LIN {X 0,Y 136.603,Z 356.091,A -85,B 0,C 180,E1 -24831.12,E2 -24831.12} C_VEL
LIN {X 0,Y 137.128,Z 356.027,A -85,B 0,C 180,E1 -24839.999,E2 -24839.999} C_VEL
LIN {X 0,Y 136.602,Z 356.09,A -85,B 0,C 180,E1 -24848.878,E2 -24848.878} C_VEL
LIN {X 0,Y 136.486,Z 356.105,A -85,B 0,C 180,E1 -24851.958,E2 -24851.958} C_VEL
LIN {X 0,Y 136.245,Z 356.134,A -85,B 0,C 180,E1 -24858.028,E2 -24858.028} C_VEL
LIN {X 0,Y 136.192,Z 356.144,A -85,B 0,C 180,E1 -24861.749,E2 -24861.749} C_VEL
LIN {X 0,Y 136.144,Z 356.148,A -85,B 0,C 180,E1 -24868.655,E2 -24868.655} C_VEL
LIN {X 0,Y 136.524,Z 356.287,A -85,B 0,C 180,E1 -24874.892,E2 -24874.892} C_VEL
LIN {X 0,Y 137.979,Z 362.492,A -85,B 0,C 180,E1 -24881.464,E2 -24881.464} C_VEL
LIN {X 0,Y 139.435,Z 367.911,A -85,B 0,C 180,E1 -24886.957,E2 -24886.957} C_VEL
LIN {X 0,Y 139.496,Z 370.039,A -85,B 0,C 180,E1 -24889.087,E2 -24889.087} C_VEL
LIN {X 0,Y 138.032,Z 374.626,A -85,B 0,C 180,E1 -24893.623,E2 -24893.623} C_VEL
LIN {X 0,Y 137.72,Z 379.074,A -85,B 0,C 180,E1 -24894.305,E2 -24894.305} C_VEL
LIN {X 0,Y 137.356,Z 394.701,A -85,B 0,C 180,E1 -24896.634,E2 -24896.634} C_VEL
LIN {X 0,Y 137.591,Z 410.054,A -85,B 0,C 180,E1 -24899.558,E2 -24899.558} C_VEL
LIN {X 0,Y 138.336,Z 425.298,A -85,B 0,C 180,E1 -24903.159,E2 -24903.159} C_VEL
LIN {X 0,Y 139.367,Z 438.842,A -85,B 0,C 180,E1 -24906.998,E2 -24906.998} C_VEL
LIN {X 0,Y 140.321,Z 447.525,A -85,B 0,C 180,E1 -24909.862,E2 -24909.862} C_VEL
LIN {X 0,Y 139.234,Z 457.776,A -85,B 0,C 180,E1 -24914.111,E2 -24914.111} C_VEL
LIN {X 0,Y 138.787,Z 467.552,A -85,B 0,C 180,E1 -24919.056,E2 -24919.056} C_VEL
LIN {X 0,Y 139.313,Z 475.809,A -85,B 0,C 180,E1 -24924.212,E2 -24924.212} C_VEL
LIN {X 0,Y 140.282,Z 481.655,A -85,B 0,C 180,E1 -24928.711,E2 -24928.711} C_VEL
LIN {X 0,Y 140.568,Z 483.669,A -85,B 0,C 180,E1 -24930.647,E2 -24930.647} C_VEL
LIN {X 0,Y 139.909,Z 485.281,A -85,B 0,C 180,E1 -24932.882,E2 -24932.882} C_VEL
LIN {X 0,Y 137.869,Z 488.121,A -85,B 0,C 180,E1 -24938.799,E2 -24938.799} C_VEL
LIN {X 0,Y 137.224,Z 489.871,A -85,B 0,C 180,E1 -24944.84,E2 -24944.84} C_VEL
LIN {X 0,Y 138.316,Z 490.738,A -85,B 0,C 180,E1 -24950.838,E2 -24950.838} C_VEL
LIN {X 0,Y 141.251,Z 490.873,A -85,B 0,C 180,E1 -24956.605,E2 -24956.605} C_VEL
LIN {X 0,Y 148.821,Z 489.76,A -85,B 0,C 180,E1 -24964.523,E2 -24964.523} C_VEL
LIN {X 0,Y 159.675,Z 487.114,A -85,B 0,C 180,E1 -24971.319,E2 -24971.319} C_VEL
LIN {X 0,Y 168.489,Z 484.531,A -85,B 0,C 180,E1 -24975.165,E2 -24975.165} C_VEL
LIN {X 0,Y 181.11,Z 480.199,A -85,B 0,C 180,E1 -24979.582,E2 -24979.582} C_VEL
LIN {X 0,Y 181.549,Z 479.751,A -85,B 0,C 180,E1 -24980.201,E2 -24980.201} C_VEL
LIN {X 0,Y 174.225,Z 479.446,A -85,B 0,C 180,E1 -24982.766,E2 -24982.766} C_VEL
LIN {X 0,Y 162.472,Z 477.5,A -85,B 0,C 180,E1 -24987.929,E2 -24987.929} C_VEL
LIN {X 0,Y 154.17,Z 474.585,A -85,B 0,C 180,E1 -24992.88,E2 -24992.88} C_VEL
LIN {X 0,Y 147.888,Z 470.965,A -85,B 0,C 180,E1 -24997.702,E2 -24997.702} C_VEL
LIN {X 0,Y 145.198,Z 469.279,A -85,B 0,C 180,E1 -24999.639,E2 -24999.639} C_VEL
LIN {X 0,Y 139.454,Z 466.109,A -85,B 0,C 180,E1 -25002.635,E2 -25002.635} C_VEL
LIN {X 0,Y 134.168,Z 462.429,A -85,B 0,C 180,E1 -25005.808,E2 -25005.808} C_VEL
LIN {X 0,Y 132.282,Z 459.913,A -85,B 0,C 180,E1 -25007.973,E2 -25007.973} C_VEL
LIN {X 0,Y 129.903,Z 451.969,A -85,B 0,C 180,E1 -25014.568,E2 -25014.568} C_VEL
LIN {X 0,Y 129.082,Z 443.16,A -85,B 0,C 180,E1 -25020.781,E2 -25020.781} C_VEL
LIN {X 0,Y 129.146,Z 432.525,A -85,B 0,C 180,E1 -25027.034,E2 -25027.034} C_VEL
LIN {X 0,Y 130.087,Z 423.208,A -85,B 0,C 180,E1 -25031.69,E2 -25031.69} C_VEL
LIN {X 0,Y 131.579,Z 412.383,A -85,B 0,C 180,E1 -25036.286,E2 -25036.286} C_VEL
LIN {X 0,Y 133.527,Z 399.543,A -85,B 0,C 180,E1 -25040.811,E2 -25040.811} C_VEL
LIN {X 0,Y 135.909,Z 385.871,A -85,B 0,C 180,E1 -25044.78,E2 -25044.78} C_VEL
LIN {X 0,Y 135.967,Z 384.573,A -85,B 0,C 180,E1 -25045.112,E2 -25045.112} C_VEL
LIN {X 0,Y 132.484,Z 371.01,A -85,B 0,C 180,E1 -25048.519,E2 -25048.519} C_VEL
LIN {X 0,Y 129.268,Z 357.522,A -85,B 0,C 180,E1 -25051.607,E2 -25051.607} C_VEL
LIN {X 0,Y 129.144,Z 357.047,A -85,B 0,C 180,E1 -25052.223,E2 -25052.223} C_VEL
LIN {X 0,Y 128.941,Z 357.043,A -85,B 0,C 180,E1 -25056.84,E2 -25056.84} C_VEL
LIN {X 0,Y 128.951,Z 357.047,A -85,B 0,C 180,E1 -25060.847,E2 -25060.847} C_VEL
LIN {X 0,Y 128.931,Z 357.043,A -85,B 0,C 180,E1 -25065.125,E2 -25065.125} C_VEL
LIN {X 0,Y 128.965,Z 357.045,A -85,B 0,C 180,E1 -25069.725,E2 -25069.725} C_VEL
LIN {X 0,Y 128.998,Z 357.038,A -85,B 0,C 180,E1 -25074.809,E2 -25074.809} C_VEL
LIN {X 0,Y 129.022,Z 357.034,A -85,B 0,C 180,E1 -25080.64,E2 -25080.64} C_VEL
LIN {X 0,Y 129.032,Z 357.035,A -85,B 0,C 180,E1 -25084.165,E2 -25084.165} C_VEL
LIN {X 0,Y 129.112,Z 357.027,A -85,B 0,C 180,E1 -25087.726,E2 -25087.726} C_VEL
LIN {X 0,Y 129.164,Z 357.014,A -85,B 0,C 180,E1 -25090.943,E2 -25090.943} C_VEL
LIN {X 0,Y 129.423,Z 356.985,A -85,B 0,C 180,E1 -25097.813,E2 -25097.813} C_VEL
LIN {X 0,Y 129.536,Z 356.971,A -85,B 0,C 180,E1 -25100.63,E2 -25100.63} C_VEL
LIN {X 0,Y 130.094,Z 356.903,A -85,B 0,C 180,E1 -25109.997,E2 -25109.997} C_VEL
LIN {X 0,Y 129.534,Z 356.974,A -85,B 0,C 180,E1 -25119.365,E2 -25119.365} C_VEL
LIN {X 0,Y 129.397,Z 356.99,A -85,B 0,C 180,E1 -25122.545,E2 -25122.545} C_VEL
LIN {X 0,Y 129.165,Z 357.021,A -85,B 0,C 180,E1 -25129.051,E2 -25129.051} C_VEL
LIN {X 0,Y 129.109,Z 357.023,A -85,B 0,C 180,E1 -25132.395,E2 -25132.395} C_VEL
LIN {X 0,Y 129.031,Z 357.036,A -85,B 0,C 180,E1 -25135.829,E2 -25135.829} C_VEL
LIN {X 0,Y 129.016,Z 357.038,A -85,B 0,C 180,E1 -25139.355,E2 -25139.355} C_VEL
LIN {X 0,Y 128.98,Z 357.043,A -85,B 0,C 180,E1 -25145.18,E2 -25145.18} C_VEL
LIN {X 0,Y 128.932,Z 357.043,A -85,B 0,C 180,E1 -25150.848,E2 -25150.848} C_VEL
LIN {X 0,Y 128.918,Z 357.052,A -85,B 0,C 180,E1 -25155.124,E2 -25155.124} C_VEL
LIN {X 0,Y 128.939,Z 357.043,A -85,B 0,C 180,E1 -25159.732,E2 -25159.732} C_VEL
LIN {X 0,Y 128.979,Z 357.044,A -85,B 0,C 180,E1 -25164.814,E2 -25164.814} C_VEL
LIN {X 0,Y 129.046,Z 357.034,A -85,B 0,C 180,E1 -25170.649,E2 -25170.649} C_VEL
LIN {X 0,Y 129.103,Z 357.025,A -85,B 0,C 180,E1 -25177.725,E2 -25177.725} C_VEL
LIN {X 0,Y 129.158,Z 357.022,A -85,B 0,C 180,E1 -25180.944,E2 -25180.944} C_VEL
LIN {X 0,Y 129.413,Z 356.988,A -85,B 0,C 180,E1 -25187.813,E2 -25187.813} C_VEL
LIN {X 0,Y 129.525,Z 356.975,A -85,B 0,C 180,E1 -25190.631,E2 -25190.631} C_VEL
LIN {X 0,Y 130.084,Z 356.905,A -85,B 0,C 180,E1 -25199.999,E2 -25199.999} C_VEL
LIN {X 0,Y 129.524,Z 356.971,A -85,B 0,C 180,E1 -25209.368,E2 -25209.368} C_VEL
LIN {X 0,Y 129.388,Z 356.992,A -85,B 0,C 180,E1 -25212.548,E2 -25212.548} C_VEL
LIN {X 0,Y 129.153,Z 357.014,A -85,B 0,C 180,E1 -25219.055,E2 -25219.055} C_VEL
LIN {X 0,Y 129.102,Z 357.029,A -85,B 0,C 180,E1 -25222.399,E2 -25222.399} C_VEL
LIN {X 0,Y 129.097,Z 357.026,A -85,B 0,C 180,E1 -25229.427,E2 -25229.427} C_VEL
LIN {X 0,Y 129.494,Z 357.096,A -85,B 0,C 180,E1 -25235.283,E2 -25235.283} C_VEL
LIN {X 0,Y 130.801,Z 362.398,A -85,B 0,C 180,E1 -25241.221,E2 -25241.221} C_VEL
LIN {X 0,Y 132.11,Z 367.066,A -85,B 0,C 180,E1 -25246.25,E2 -25246.25} C_VEL
LIN {X 0,Y 132.475,Z 368.687,A -85,B 0,C 180,E1 -25247.963,E2 -25247.963} C_VEL
LIN {X 0,Y 131.943,Z 370.854,A -85,B 0,C 180,E1 -25250.273,E2 -25250.273} C_VEL
LIN {X 0,Y 131.065,Z 373.682,A -85,B 0,C 180,E1 -25253.166,E2 -25253.166} C_VEL
LIN {X 0,Y 130.265,Z 391.666,A -85,B 0,C 180,E1 -25255.965,E2 -25255.965} C_VEL
LIN {X 0,Y 130.43,Z 406.961,A -85,B 0,C 180,E1 -25258.967,E2 -25258.967} C_VEL
LIN {X 0,Y 131.047,Z 421.405,A -85,B 0,C 180,E1 -25262.451,E2 -25262.451} C_VEL
LIN {X 0,Y 132.042,Z 435.246,A -85,B 0,C 180,E1 -25266.476,E2 -25266.476} C_VEL
LIN {X 0,Y 133.341,Z 446.662,A -85,B 0,C 180,E1 -25270.369,E2 -25270.369} C_VEL
LIN {X 0,Y 132.394,Z 456.294,A -85,B 0,C 180,E1 -25274.611,E2 -25274.611} C_VEL
LIN {X 0,Y 132.062,Z 465.103,A -85,B 0,C 180,E1 -25279.268,E2 -25279.268} C_VEL
LIN {X 0,Y 132.653,Z 473.561,A -85,B 0,C 180,E1 -25284.683,E2 -25284.683} C_VEL
LIN {X 0,Y 133.563,Z 478.708,A -85,B 0,C 180,E1 -25288.73,E2 -25288.73} C_VEL
LIN {X 0,Y 133.876,Z 480.168,A -85,B 0,C 180,E1 -25290.003,E2 -25290.003} C_VEL
LIN {X 0,Y 133.296,Z 482.552,A -85,B 0,C 180,E1 -25293.025,E2 -25293.025} C_VEL
LIN {X 0,Y 131.23,Z 485.546,A -85,B 0,C 180,E1 -25299.248,E2 -25299.248} C_VEL
LIN {X 0,Y 130.635,Z 487.479,A -85,B 0,C 180,E1 -25305.607,E2 -25305.607} C_VEL
LIN {X 0,Y 131.911,Z 488.565,A -85,B 0,C 180,E1 -25311.9,E2 -25311.9} C_VEL
LIN {X 0,Y 135.079,Z 488.926,A -85,B 0,C 180,E1 -25317.924,E2 -25317.924} C_VEL
LIN {X 0,Y 140.013,Z 488.576,A -85,B 0,C 180,E1 -25323.517,E2 -25323.517} C_VEL
LIN {X 0,Y 146.563,Z 487.63,A -85,B 0,C 180,E1 -25328.566,E2 -25328.566} C_VEL
LIN {X 0,Y 158.864,Z 484.979,A -85,B 0,C 180,E1 -25335.061,E2 -25335.061} C_VEL
LIN {X 0,Y 171.356,Z 481.571,A -85,B 0,C 180,E1 -25339.656,E2 -25339.656} C_VEL
LIN {X 0,Y 170.756,Z 481.068,A -85,B 0,C 180,E1 -25340.61,E2 -25340.61} C_VEL
LIN {X 0,Y 159.635,Z 479.231,A -85,B 0,C 180,E1 -25345.088,E2 -25345.088} C_VEL
LIN {X 0,Y 151.563,Z 476.711,A -85,B 0,C 180,E1 -25349.332,E2 -25349.332} C_VEL
LIN {X 0,Y 142.923,Z 472.226,A -85,B 0,C 180,E1 -25355.294,E2 -25355.294} C_VEL
LIN {X 0,Y 136.232,Z 466.215,A -85,B 0,C 180,E1 -25361.97,E2 -25361.97} C_VEL
LIN {X 0,Y 132.282,Z 459.913,A -85,B 0,C 180,E1 -25367.973,E2 -25367.973} C_VEL
LIN {X 0,Y 130.663,Z 457.299,A -85,B 0,C 180,E1 -25370.158,E2 -25370.158} C_VEL
LIN {X 0,Y 126.723,Z 452.536,A -85,B 0,C 180,E1 -25373.598,E2 -25373.598} C_VEL
LIN {X 0,Y 123.152,Z 447.252,A -85,B 0,C 180,E1 -25377.117,E2 -25377.117} C_VEL
LIN {X 0,Y 122.177,Z 443.872,A -85,B 0,C 180,E1 -25379.36,E2 -25379.36} C_VEL
LIN {X 0,Y 121.971,Z 433.547,A -85,B 0,C 180,E1 -25385.788,E2 -25385.788} C_VEL
LIN {X 0,Y 122.985,Z 423.193,A -85,B 0,C 180,E1 -25391.256,E2 -25391.256} C_VEL
LIN {X 0,Y 124.542,Z 411.592,A -85,B 0,C 180,E1 -25396.39,E2 -25396.39} C_VEL
LIN {X 0,Y 126.539,Z 398.546,A -85,B 0,C 180,E1 -25401.163,E2 -25401.163} C_VEL
LIN {X 0,Y 128.82,Z 385.674,A -85,B 0,C 180,E1 -25405.013,E2 -25405.013} C_VEL
LIN {X 0,Y 125.748,Z 373.225,A -85,B 0,C 180,E1 -25408.323,E2 -25408.323} C_VEL
LIN {X 0,Y 122.197,Z 358.436,A -85,B 0,C 180,E1 -25411.898,E2 -25411.898} C_VEL
LIN {X 0,Y 122.095,Z 357.915,A -85,B 0,C 180,E1 -25412.658,E2 -25412.658} C_VEL
LIN {X 0,Y 121.87,Z 357.928,A -85,B 0,C 180,E1 -25419.373,E2 -25419.373} C_VEL
LIN {X 0,Y 121.855,Z 357.928,A -85,B 0,C 180,E1 -25423.798,E2 -25423.798} C_VEL
LIN {X 0,Y 121.892,Z 357.927,A -85,B 0,C 180,E1 -25428.553,E2 -25428.553} C_VEL
LIN {X 0,Y 121.951,Z 357.915,A -85,B 0,C 180,E1 -25434.806,E2 -25434.806} C_VEL
LIN {X 0,Y 121.935,Z 357.92,A -85,B 0,C 180,E1 -25439.835,E2 -25439.835} C_VEL
LIN {X 0,Y 121.987,Z 357.916,A -85,B 0,C 180,E1 -25446.213,E2 -25446.213} C_VEL
LIN {X 0,Y 122.054,Z 357.901,A -85,B 0,C 180,E1 -25449.785,E2 -25449.785} C_VEL
LIN {X 0,Y 122.269,Z 357.878,A -85,B 0,C 180,E1 -25456.705,E2 -25456.705} C_VEL
LIN {X 0,Y 122.462,Z 357.85,A -85,B 0,C 180,E1 -25460.083,E2 -25460.083} C_VEL
LIN {X 0,Y 122.614,Z 357.832,A -85,B 0,C 180,E1 -25466.711,E2 -25466.711} C_VEL
LIN {X 0,Y 123.048,Z 357.781,A -85,B 0,C 180,E1 -25469.997,E2 -25469.997} C_VEL
LIN {X 0,Y 122.459,Z 357.849,A -85,B 0,C 180,E1 -25476.588,E2 -25476.588} C_VEL
LIN {X 0,Y 122.46,Z 357.856,A -85,B 0,C 180,E1 -25479.911,E2 -25479.911} C_VEL
LIN {X 0,Y 122.267,Z 357.877,A -85,B 0,C 180,E1 -25483.289,E2 -25483.289} C_VEL
LIN {X 0,Y 122.053,Z 357.905,A -85,B 0,C 180,E1 -25490.208,E2 -25490.208} C_VEL
LIN {X 0,Y 121.984,Z 357.909,A -85,B 0,C 180,E1 -25493.781,E2 -25493.781} C_VEL
LIN {X 0,Y 121.928,Z 357.919,A -85,B 0,C 180,E1 -25500.16,E2 -25500.16} C_VEL
LIN {X 0,Y 121.898,Z 357.925,A -85,B 0,C 180,E1 -25506.178,E2 -25506.178} C_VEL
LIN {X 0,Y 121.87,Z 357.924,A -85,B 0,C 180,E1 -25511.436,E2 -25511.436} C_VEL
LIN {X 0,Y 121.869,Z 357.924,A -85,B 0,C 180,E1 -25518.558,E2 -25518.558} C_VEL
LIN {X 0,Y 121.931,Z 357.921,A -85,B 0,C 180,E1 -25524.802,E2 -25524.802} C_VEL
LIN {X 0,Y 121.937,Z 357.918,A -85,B 0,C 180,E1 -25529.824,E2 -25529.824} C_VEL
LIN {X 0,Y 121.979,Z 357.909,A -85,B 0,C 180,E1 -25536.213,E2 -25536.213} C_VEL
LIN {X 0,Y 122.046,Z 357.906,A -85,B 0,C 180,E1 -25539.786,E2 -25539.786} C_VEL
LIN {X 0,Y 122.26,Z 357.878,A -85,B 0,C 180,E1 -25546.706,E2 -25546.706} C_VEL
LIN {X 0,Y 122.451,Z 357.857,A -85,B 0,C 180,E1 -25550.084,E2 -25550.084} C_VEL
LIN {X 0,Y 122.605,Z 357.838,A -85,B 0,C 180,E1 -25556.713,E2 -25556.713} C_VEL
LIN {X 0,Y 123.038,Z 357.782,A -85,B 0,C 180,E1 -25559.999,E2 -25559.999} C_VEL
LIN {X 0,Y 122.45,Z 357.857,A -85,B 0,C 180,E1 -25566.591,E2 -25566.591} C_VEL
LIN {X 0,Y 122.45,Z 357.851,A -85,B 0,C 180,E1 -25569.914,E2 -25569.914} C_VEL
LIN {X 0,Y 122.258,Z 357.879,A -85,B 0,C 180,E1 -25573.293,E2 -25573.293} C_VEL
LIN {X 0,Y 122.043,Z 357.903,A -85,B 0,C 180,E1 -25580.213,E2 -25580.213} C_VEL
LIN {X 0,Y 121.978,Z 357.917,A -85,B 0,C 180,E1 -25583.785,E2 -25583.785} C_VEL
LIN {X 0,Y 122.078,Z 357.903,A -85,B 0,C 180,E1 -25591.206,E2 -25591.206} C_VEL
LIN {X 0,Y 122.496,Z 357.946,A -85,B 0,C 180,E1 -25595.868,E2 -25595.868} C_VEL
LIN {X 0,Y 124.059,Z 363.872,A -85,B 0,C 180,E1 -25602.828,E2 -25602.828} C_VEL
LIN {X 0,Y 125.274,Z 368.163,A -85,B 0,C 180,E1 -25607.689,E2 -25607.689} C_VEL
LIN {X 0,Y 124.989,Z 369.943,A -85,B 0,C 180,E1 -25609.716,E2 -25609.716} C_VEL
LIN {X 0,Y 124.089,Z 372.745,A -85,B 0,C 180,E1 -25612.704,E2 -25612.704} C_VEL
LIN {X 0,Y 123.219,Z 389.789,A -85,B 0,C 180,E1 -25615.491,E2 -25615.491} C_VEL
LIN {X 0,Y 123.305,Z 405.547,A -85,B 0,C 180,E1 -25618.753,E2 -25618.753} C_VEL
LIN {X 0,Y 123.878,Z 418.797,A -85,B 0,C 180,E1 -25622.096,E2 -25622.096} C_VEL
LIN {X 0,Y 124.848,Z 432.037,A -85,B 0,C 180,E1 -25626.073,E2 -25626.073} C_VEL
LIN {X 0,Y 126.355,Z 444.58,A -85,B 0,C 180,E1 -25630.508,E2 -25630.508} C_VEL
LIN {X 0,Y 125.677,Z 453.596,A -85,B 0,C 180,E1 -25634.599,E2 -25634.599} C_VEL
LIN {X 0,Y 125.369,Z 462.556,A -85,B 0,C 180,E1 -25639.506,E2 -25639.506} C_VEL
LIN {X 0,Y 126.046,Z 471.181,A -85,B 0,C 180,E1 -25645.205,E2 -25645.205} C_VEL
LIN {X 0,Y 127.183,Z 477.053,A -85,B 0,C 180,E1 -25650.003,E2 -25650.003} C_VEL
LIN {X 0,Y 127.128,Z 479.003,A -85,B 0,C 180,E1 -25652.137,E2 -25652.137} C_VEL
LIN {X 0,Y 125.538,Z 481.421,A -85,B 0,C 180,E1 -25656.432,E2 -25656.432} C_VEL
LIN {X 0,Y 124.145,Z 484.024,A -85,B 0,C 180,E1 -25663.091,E2 -25663.091} C_VEL
LIN {X 0,Y 125.566,Z 486.272,A -85,B 0,C 180,E1 -25673.069,E2 -25673.069} C_VEL
LIN {X 0,Y 131.414,Z 486.873,A -85,B 0,C 180,E1 -25682.333,E2 -25682.333} C_VEL
LIN {X 0,Y 141.162,Z 486.044,A -85,B 0,C 180,E1 -25690.336,E2 -25690.336} C_VEL
LIN {X 0,Y 151.835,Z 484.281,A -85,B 0,C 180,E1 -25696.029,E2 -25696.029} C_VEL
LIN {X 0,Y 160.67,Z 482.448,A -85,B 0,C 180,E1 -25699.412,E2 -25699.412} C_VEL
LIN {X 0,Y 161.702,Z 481.829,A -85,B 0,C 180,E1 -25700.417,E2 -25700.417} C_VEL
LIN {X 0,Y 149.542,Z 478.811,A -85,B 0,C 180,E1 -25705.671,E2 -25705.671} C_VEL
LIN {X 0,Y 139.9,Z 474.457,A -85,B 0,C 180,E1 -25711.495,E2 -25711.495} C_VEL
LIN {X 0,Y 132.089,Z 468.633,A -85,B 0,C 180,E1 -25718.134,E2 -25718.134} C_VEL
LIN {X 0,Y 127.318,Z 462.817,A -85,B 0,C 180,E1 -25723.979,E2 -25723.979} C_VEL
LIN {X 0,Y 124.094,Z 455.854,A -85,B 0,C 180,E1 -25730.219,E2 -25730.219} C_VEL
LIN {X 0,Y 122.424,Z 447.597,A -85,B 0,C 180,E1 -25736.71,E2 -25736.71} C_VEL
LIN {X 0,Y 122.177,Z 443.872,A -85,B 0,C 180,E1 -25739.36,E2 -25739.36} C_VEL
LIN {X 0,Y 121.347,Z 440.448,A -85,B 0,C 180,E1 -25741.551,E2 -25741.551} C_VEL
LIN {X 0,Y 118.608,Z 434.253,A -85,B 0,C 180,E1 -25744.993,E2 -25744.993} C_VEL
LIN {X 0,Y 116.159,Z 427.641,A -85,B 0,C 180,E1 -25748.439,E2 -25748.439} C_VEL
LIN {X 0,Y 115.837,Z 423.476,A -85,B 0,C 180,E1 -25750.559,E2 -25750.559} C_VEL
LIN {X 0,Y 117.373,Z 411.494,A -85,B 0,C 180,E1 -25756.155,E2 -25756.155} C_VEL
LIN {X 0,Y 119.409,Z 398.529,A -85,B 0,C 180,E1 -25761.132,E2 -25761.132} C_VEL
LIN {X 0,Y 121.588,Z 385.463,A -85,B 0,C 180,E1 -25765.233,E2 -25765.233} C_VEL
LIN {X 0,Y 117.891,Z 370.949,A -85,B 0,C 180,E1 -25769.229,E2 -25769.229} C_VEL
LIN {X 0,Y 115.161,Z 359.392,A -85,B 0,C 180,E1 -25772.124,E2 -25772.124} C_VEL
LIN {X 0,Y 115.043,Z 358.81,A -85,B 0,C 180,E1 -25772.806,E2 -25772.806} C_VEL
LIN {X 0,Y 114.795,Z 358.806,A -85,B 0,C 180,E1 -25777.752,E2 -25777.752} C_VEL
LIN {X 0,Y 114.799,Z 358.808,A -85,B 0,C 180,E1 -25782.719,E2 -25782.719} C_VEL
LIN {X 0,Y 114.811,Z 358.807,A -85,B 0,C 180,E1 -25787.67,E2 -25787.67} C_VEL
LIN {X 0,Y 114.818,Z 358.801,A -85,B 0,C 180,E1 -25792.726,E2 -25792.726} C_VEL
LIN {X 0,Y 114.869,Z 358.8,A -85,B 0,C 180,E1 -25798.934,E2 -25798.934} C_VEL
LIN {X 0,Y 114.952,Z 358.791,A -85,B 0,C 180,E1 -25806.505,E2 -25806.505} C_VEL
LIN {X 0,Y 115.023,Z 358.778,A -85,B 0,C 180,E1 -25812.208,E2 -25812.208} C_VEL
LIN {X 0,Y 115.291,Z 358.747,A -85,B 0,C 180,E1 -25817.255,E2 -25817.255} C_VEL
LIN {X 0,Y 115.398,Z 358.728,A -85,B 0,C 180,E1 -25819.469,E2 -25819.469} C_VEL
LIN {X 0,Y 115.541,Z 358.713,A -85,B 0,C 180,E1 -25826.51,E2 -25826.51} C_VEL
LIN {X 0,Y 116,Z 358.658,A -85,B 0,C 180,E1 -25829.997,E2 -25829.997} C_VEL
LIN {X 0,Y 115.401,Z 358.728,A -85,B 0,C 180,E1 -25836.993,E2 -25836.993} C_VEL
LIN {X 0,Y 115.396,Z 358.735,A -85,B 0,C 180,E1 -25840.524,E2 -25840.524} C_VEL
LIN {X 0,Y 115.151,Z 358.76,A -85,B 0,C 180,E1 -25844.127,E2 -25844.127} C_VEL
LIN {X 0,Y 114.985,Z 358.784,A -85,B 0,C 180,E1 -25851.51,E2 -25851.51} C_VEL
LIN {X 0,Y 114.868,Z 358.798,A -85,B 0,C 180,E1 -25855.355,E2 -25855.355} C_VEL
LIN {X 0,Y 114.861,Z 358.797,A -85,B 0,C 180,E1 -25861.059,E2 -25861.059} C_VEL
LIN {X 0,Y 114.787,Z 358.81,A -85,B 0,C 180,E1 -25867.749,E2 -25867.749} C_VEL
LIN {X 0,Y 114.785,Z 358.809,A -85,B 0,C 180,E1 -25872.714,E2 -25872.714} C_VEL
LIN {X 0,Y 114.792,Z 358.807,A -85,B 0,C 180,E1 -25877.664,E2 -25877.664} C_VEL
LIN {X 0,Y 114.796,Z 358.81,A -85,B 0,C 180,E1 -25882.733,E2 -25882.733} C_VEL
LIN {X 0,Y 114.864,Z 358.797,A -85,B 0,C 180,E1 -25888.93,E2 -25888.93} C_VEL
LIN {X 0,Y 114.942,Z 358.785,A -85,B 0,C 180,E1 -25896.505,E2 -25896.505} C_VEL
LIN {X 0,Y 115.015,Z 358.783,A -85,B 0,C 180,E1 -25902.209,E2 -25902.209} C_VEL
LIN {X 0,Y 115.281,Z 358.749,A -85,B 0,C 180,E1 -25907.256,E2 -25907.256} C_VEL
LIN {X 0,Y 115.387,Z 358.736,A -85,B 0,C 180,E1 -25909.471,E2 -25909.471} C_VEL
LIN {X 0,Y 115.531,Z 358.719,A -85,B 0,C 180,E1 -25916.511,E2 -25916.511} C_VEL
LIN {X 0,Y 115.99,Z 358.659,A -85,B 0,C 180,E1 -25919.999,E2 -25919.999} C_VEL
LIN {X 0,Y 115.391,Z 358.735,A -85,B 0,C 180,E1 -25926.996,E2 -25926.996} C_VEL
LIN {X 0,Y 115.387,Z 358.73,A -85,B 0,C 180,E1 -25930.528,E2 -25930.528} C_VEL
LIN {X 0,Y 115.142,Z 358.768,A -85,B 0,C 180,E1 -25934.131,E2 -25934.131} C_VEL
LIN {X 0,Y 114.975,Z 358.786,A -85,B 0,C 180,E1 -25941.515,E2 -25941.515} C_VEL
LIN {X 0,Y 114.945,Z 358.788,A -85,B 0,C 180,E1 -25949.283,E2 -25949.283} C_VEL
LIN {X 0,Y 115.542,Z 358.831,A -85,B 0,C 180,E1 -25956.644,E2 -25956.644} C_VEL
LIN {X 0,Y 117.198,Z 364.745,A -85,B 0,C 180,E1 -25963.983,E2 -25963.983} C_VEL
LIN {X 0,Y 118.061,Z 367.502,A -85,B 0,C 180,E1 -25967.275,E2 -25967.275} C_VEL
LIN {X 0,Y 117.979,Z 368.975,A -85,B 0,C 180,E1 -25969.064,E2 -25969.064} C_VEL
LIN {X 0,Y 117.129,Z 371.717,A -85,B 0,C 180,E1 -25972.185,E2 -25972.185} C_VEL
LIN {X 0,Y 116.125,Z 390.044,A -85,B 0,C 180,E1 -25975.436,E2 -25975.436} C_VEL
LIN {X 0,Y 116.21,Z 405.08,A -85,B 0,C 180,E1 -25978.793,E2 -25978.793} C_VEL
LIN {X 0,Y 116.886,Z 419.636,A -85,B 0,C 180,E1 -25982.777,E2 -25982.777} C_VEL
LIN {X 0,Y 118.001,Z 433.198,A -85,B 0,C 180,E1 -25987.227,E2 -25987.227} C_VEL
LIN {X 0,Y 119.468,Z 443.707,A -85,B 0,C 180,E1 -25991.217,E2 -25991.217} C_VEL
LIN {X 0,Y 118.867,Z 452.41,A -85,B 0,C 180,E1 -25995.45,E2 -25995.45} C_VEL
LIN {X 0,Y 118.728,Z 461.287,A -85,B 0,C 180,E1 -26000.635,E2 -26000.635} C_VEL
LIN {X 0,Y 119.631,Z 469.815,A -85,B 0,C 180,E1 -26006.635,E2 -26006.635} C_VEL
LIN {X 0,Y 120.512,Z 473.84,A -85,B 0,C 180,E1 -26010.003,E2 -26010.003} C_VEL
LIN {X 0,Y 120.619,Z 476.129,A -85,B 0,C 180,E1 -26012.488,E2 -26012.488} C_VEL
LIN {X 0,Y 119.014,Z 478.497,A -85,B 0,C 180,E1 -26016.786,E2 -26016.786} C_VEL
LIN {X 0,Y 117.643,Z 481.293,A -85,B 0,C 180,E1 -26023.828,E2 -26023.828} C_VEL
LIN {X 0,Y 118.248,Z 483.15,A -85,B 0,C 180,E1 -26030.895,E2 -26030.895} C_VEL
LIN {X 0,Y 120.971,Z 484.318,A -85,B 0,C 180,E1 -26037.699,E2 -26037.699} C_VEL
LIN {X 0,Y 128.691,Z 484.775,A -85,B 0,C 180,E1 -26046.925,E2 -26046.925} C_VEL
LIN {X 0,Y 140.063,Z 483.886,A -85,B 0,C 180,E1 -26054.63,E2 -26054.63} C_VEL
LIN {X 0,Y 150.91,Z 482.32,A -85,B 0,C 180,E1 -26059.501,E2 -26059.501} C_VEL
LIN {X 0,Y 151.707,Z 481.773,A -85,B 0,C 180,E1 -26060.553,E2 -26060.553} C_VEL
LIN {X 0,Y 143.768,Z 479.307,A -85,B 0,C 180,E1 -26064.084,E2 -26064.084} C_VEL
LIN {X 0,Y 133.714,Z 474.546,A -85,B 0,C 180,E1 -26070.046,E2 -26070.046} C_VEL
LIN {X 0,Y 125.537,Z 468.298,A -85,B 0,C 180,E1 -26076.929,E2 -26076.929} C_VEL
LIN {X 0,Y 120.534,Z 462.141,A -85,B 0,C 180,E1 -26083.051,E2 -26083.051} C_VEL
LIN {X 0,Y 116.899,Z 453.816,A -85,B 0,C 180,E1 -26090.484,E2 -26090.484} C_VEL
LIN {X 0,Y 115.298,Z 443.812,A -85,B 0,C 180,E1 -26098.254,E2 -26098.254} C_VEL
LIN {X 0,Y 114.952,Z 433.045,A -85,B 0,C 180,E1 -26105.263,E2 -26105.263} C_VEL
LIN {X 0,Y 115.837,Z 423.476,A -85,B 0,C 180,E1 -26110.559,E2 -26110.559} C_VEL
LIN {X 0,Y 115.61,Z 419.264,A -85,B 0,C 180,E1 -26112.602,E2 -26112.602} C_VEL
LIN {X 0,Y 113.739,Z 411.934,A -85,B 0,C 180,E1 -26115.794,E2 -26115.794} C_VEL
LIN {X 0,Y 112.043,Z 404.218,A -85,B 0,C 180,E1 -26118.888,E2 -26118.888} C_VEL
LIN {X 0,Y 112.118,Z 399.429,A -85,B 0,C 180,E1 -26120.694,E2 -26120.694} C_VEL
LIN {X 0,Y 114.346,Z 386.674,A -85,B 0,C 180,E1 -26124.997,E2 -26124.997} C_VEL
LIN {X 0,Y 113.506,Z 382.445,A -85,B 0,C 180,E1 -26126.29,E2 -26126.29} C_VEL
LIN {X 0,Y 109.686,Z 367.249,A -85,B 0,C 180,E1 -26130.516,E2 -26130.516} C_VEL
LIN {X 0,Y 108.121,Z 360.193,A -85,B 0,C 180,E1 -26132.427,E2 -26132.427} C_VEL
LIN {X 0,Y 107.978,Z 359.683,A -85,B 0,C 180,E1 -26133.188,E2 -26133.188} C_VEL
LIN {X 0,Y 107.693,Z 359.696,A -85,B 0,C 180,E1 -26140.739,E2 -26140.739} C_VEL
LIN {X 0,Y 107.691,Z 359.689,A -85,B 0,C 180,E1 -26145.88,E2 -26145.88} C_VEL
LIN {X 0,Y 107.715,Z 359.691,A -85,B 0,C 180,E1 -26151.534,E2 -26151.534} C_VEL
LIN {X 0,Y 107.808,Z 359.681,A -85,B 0,C 180,E1 -26158.562,E2 -26158.562} C_VEL
LIN {X 0,Y 107.917,Z 359.667,A -85,B 0,C 180,E1 -26166.996,E2 -26166.996} C_VEL
LIN {X 0,Y 108.045,Z 359.651,A -85,B 0,C 180,E1 -26174.915,E2 -26174.915} C_VEL
LIN {X 0,Y 108.311,Z 359.611,A -85,B 0,C 180,E1 -26178.772,E2 -26178.772} C_VEL
LIN {X 0,Y 108.467,Z 359.594,A -85,B 0,C 180,E1 -26186.282,E2 -26186.282} C_VEL
LIN {X 0,Y 108.951,Z 359.536,A -85,B 0,C 180,E1 -26189.997,E2 -26189.997} C_VEL
LIN {X 0,Y 108.343,Z 359.608,A -85,B 0,C 180,E1 -26197.451,E2 -26197.451} C_VEL
LIN {X 0,Y 108.205,Z 359.629,A -85,B 0,C 180,E1 -26203.022,E2 -26203.022} C_VEL
LIN {X 0,Y 107.912,Z 359.668,A -85,B 0,C 180,E1 -26209,E2 -26209} C_VEL
LIN {X 0,Y 107.857,Z 359.669,A -85,B 0,C 180,E1 -26214.18,E2 -26214.18} C_VEL
LIN {X 0,Y 107.787,Z 359.676,A -85,B 0,C 180,E1 -26222.042,E2 -26222.042} C_VEL
LIN {X 0,Y 107.694,Z 359.693,A -85,B 0,C 180,E1 -26228.452,E2 -26228.452} C_VEL
LIN {X 0,Y 107.674,Z 359.697,A -85,B 0,C 180,E1 -26235.883,E2 -26235.883} C_VEL
LIN {X 0,Y 107.693,Z 359.694,A -85,B 0,C 180,E1 -26241.541,E2 -26241.541} C_VEL
LIN {X 0,Y 107.801,Z 359.675,A -85,B 0,C 180,E1 -26248.562,E2 -26248.562} C_VEL
LIN {X 0,Y 107.906,Z 359.662,A -85,B 0,C 180,E1 -26256.996,E2 -26256.996} C_VEL
LIN {X 0,Y 108.035,Z 359.646,A -85,B 0,C 180,E1 -26264.916,E2 -26264.916} C_VEL
LIN {X 0,Y 108.301,Z 359.62,A -85,B 0,C 180,E1 -26268.773,E2 -26268.773} C_VEL
LIN {X 0,Y 108.457,Z 359.599,A -85,B 0,C 180,E1 -26276.284,E2 -26276.284} C_VEL
LIN {X 0,Y 108.941,Z 359.537,A -85,B 0,C 180,E1 -26279.999,E2 -26279.999} C_VEL
LIN {X 0,Y 108.334,Z 359.615,A -85,B 0,C 180,E1 -26287.454,E2 -26287.454} C_VEL
LIN {X 0,Y 108.197,Z 359.631,A -85,B 0,C 180,E1 -26293.025,E2 -26293.025} C_VEL
LIN {X 0,Y 107.902,Z 359.661,A -85,B 0,C 180,E1 -26299.005,E2 -26299.005} C_VEL
LIN {X 0,Y 107.856,Z 359.675,A -85,B 0,C 180,E1 -26304.191,E2 -26304.191} C_VEL
LIN {X 0,Y 108.04,Z 359.652,A -85,B 0,C 180,E1 -26312.266,E2 -26312.266} C_VEL
LIN {X 0,Y 108.641,Z 359.723,A -85,B 0,C 180,E1 -26317.626,E2 -26317.626} C_VEL
LIN {X 0,Y 110.199,Z 364.975,A -85,B 0,C 180,E1 -26324.549,E2 -26324.549} C_VEL
LIN {X 0,Y 110.947,Z 367.679,A -85,B 0,C 180,E1 -26327.989,E2 -26327.989} C_VEL
LIN {X 0,Y 110.184,Z 370.692,A -85,B 0,C 180,E1 -26331.696,E2 -26331.696} C_VEL
LIN {X 0,Y 109.166,Z 386.383,A -85,B 0,C 180,E1 -26334.595,E2 -26334.595} C_VEL
LIN {X 0,Y 109.04,Z 400.994,A -85,B 0,C 180,E1 -26337.957,E2 -26337.957} C_VEL
LIN {X 0,Y 109.663,Z 416.43,A -85,B 0,C 180,E1 -26342.317,E2 -26342.317} C_VEL
LIN {X 0,Y 110.74,Z 429.214,A -85,B 0,C 180,E1 -26346.635,E2 -26346.635} C_VEL
LIN {X 0,Y 112.507,Z 442.211,A -85,B 0,C 180,E1 -26351.804,E2 -26351.804} C_VEL
LIN {X 0,Y 112.286,Z 447.785,A -85,B 0,C 180,E1 -26354.577,E2 -26354.577} C_VEL
LIN {X 0,Y 112.057,Z 457.192,A -85,B 0,C 180,E1 -26360.072,E2 -26360.072} C_VEL
LIN {X 0,Y 112.925,Z 466.188,A -85,B 0,C 180,E1 -26366.435,E2 -26366.435} C_VEL
LIN {X 0,Y 113.816,Z 470.443,A -85,B 0,C 180,E1 -26370.003,E2 -26370.003} C_VEL
LIN {X 0,Y 114.214,Z 472.258,A -85,B 0,C 180,E1 -26371.766,E2 -26371.766} C_VEL
LIN {X 0,Y 113.862,Z 473.566,A -85,B 0,C 180,E1 -26373.542,E2 -26373.542} C_VEL
LIN {X 0,Y 111.664,Z 477.082,A -85,B 0,C 180,E1 -26380.887,E2 -26380.887} C_VEL
LIN {X 0,Y 111.998,Z 480.493,A -85,B 0,C 180,E1 -26392.121,E2 -26392.121} C_VEL
LIN {X 0,Y 117.303,Z 482.264,A -85,B 0,C 180,E1 -26402.634,E2 -26402.634} C_VEL
LIN {X 0,Y 126.895,Z 482.626,A -85,B 0,C 180,E1 -26411.656,E2 -26411.656} C_VEL
LIN {X 0,Y 139.831,Z 481.709,A -85,B 0,C 180,E1 -26418.934,E2 -26418.934} C_VEL
LIN {X 0,Y 142.798,Z 481.338,A -85,B 0,C 180,E1 -26420.223,E2 -26420.223} C_VEL
LIN {X 0,Y 131.61,Z 476.68,A -85,B 0,C 180,E1 -26425.896,E2 -26425.896} C_VEL
LIN {X 0,Y 122.164,Z 470.621,A -85,B 0,C 180,E1 -26432.599,E2 -26432.599} C_VEL
LIN {X 0,Y 115.007,Z 462.971,A -85,B 0,C 180,E1 -26440.361,E2 -26440.361} C_VEL
LIN {X 0,Y 110.637,Z 454.587,A -85,B 0,C 180,E1 -26448.087,E2 -26448.087} C_VEL
LIN {X 0,Y 108.511,Z 444.582,A -85,B 0,C 180,E1 -26456.287,E2 -26456.287} C_VEL
LIN {X 0,Y 107.908,Z 435.279,A -85,B 0,C 180,E1 -26462.801,E2 -26462.801} C_VEL
LIN {X 0,Y 108.636,Z 424.474,A -85,B 0,C 180,E1 -26469.309,E2 -26469.309} C_VEL
LIN {X 0,Y 110.033,Z 412.553,A -85,B 0,C 180,E1 -26475.289,E2 -26475.289} C_VEL
LIN {X 0,Y 112.118,Z 399.429,A -85,B 0,C 180,E1 -26480.694,E2 -26480.694} C_VEL
LIN {X 0,Y 112.201,Z 396.281,A -85,B 0,C 180,E1 -26481.835,E2 -26481.835} C_VEL
LIN {X 0,Y 111.185,Z 391.443,A -85,B 0,C 180,E1 -26483.493,E2 -26483.493} C_VEL
LIN {X 0,Y 109.323,Z 386.676,A -85,B 0,C 180,E1 -26485.052,E2 -26485.052} C_VEL
LIN {X 0,Y 106.336,Z 380.026,A -85,B 0,C 180,E1 -26487.159,E2 -26487.159} C_VEL
LIN {X 0,Y 103.819,Z 373.119,A -85,B 0,C 180,E1 -26489.233,E2 -26489.233} C_VEL
LIN {X 0,Y 101.045,Z 361.082,A -85,B 0,C 180,E1 -26492.655,E2 -26492.655} C_VEL
LIN {X 0,Y 100.905,Z 360.579,A -85,B 0,C 180,E1 -26493.295,E2 -26493.295} C_VEL
LIN {X 0,Y 100.653,Z 360.571,A -85,B 0,C 180,E1 -26499.814,E2 -26499.814} C_VEL
LIN {X 0,Y 100.661,Z 360.564,A -85,B 0,C 180,E1 -26505.714,E2 -26505.714} C_VEL
LIN {X 0,Y 100.652,Z 360.57,A -85,B 0,C 180,E1 -26511.062,E2 -26511.062} C_VEL
LIN {X 0,Y 100.704,Z 360.566,A -85,B 0,C 180,E1 -26516.876,E2 -26516.876} C_VEL
LIN {X 0,Y 100.791,Z 360.554,A -85,B 0,C 180,E1 -26525.265,E2 -26525.265} C_VEL
LIN {X 0,Y 100.824,Z 360.545,A -85,B 0,C 180,E1 -26529.599,E2 -26529.599} C_VEL
LIN {X 0,Y 101.204,Z 360.498,A -85,B 0,C 180,E1 -26537.972,E2 -26537.972} C_VEL
LIN {X 0,Y 101.284,Z 360.492,A -85,B 0,C 180,E1 -26542.019,E2 -26542.019} C_VEL
LIN {X 0,Y 101.875,Z 360.417,A -85,B 0,C 180,E1 -26549.996,E2 -26549.996} C_VEL
LIN {X 0,Y 101.282,Z 360.489,A -85,B 0,C 180,E1 -26557.974,E2 -26557.974} C_VEL
LIN {X 0,Y 101.131,Z 360.508,A -85,B 0,C 180,E1 -26563.36,E2 -26563.36} C_VEL
LIN {X 0,Y 100.821,Z 360.55,A -85,B 0,C 180,E1 -26570.394,E2 -26570.394} C_VEL
LIN {X 0,Y 100.774,Z 360.552,A -85,B 0,C 180,E1 -26574.954,E2 -26574.954} C_VEL
LIN {X 0,Y 100.694,Z 360.561,A -85,B 0,C 180,E1 -26583.115,E2 -26583.115} C_VEL
LIN {X 0,Y 100.643,Z 360.567,A -85,B 0,C 180,E1 -26589.811,E2 -26589.811} C_VEL
LIN {X 0,Y 100.645,Z 360.572,A -85,B 0,C 180,E1 -26595.708,E2 -26595.708} C_VEL
LIN {X 0,Y 100.63,Z 360.571,A -85,B 0,C 180,E1 -26601.055,E2 -26601.055} C_VEL
LIN {X 0,Y 100.693,Z 360.56,A -85,B 0,C 180,E1 -26606.875,E2 -26606.875} C_VEL
LIN {X 0,Y 100.781,Z 360.55,A -85,B 0,C 180,E1 -26615.264,E2 -26615.264} C_VEL
LIN {X 0,Y 100.814,Z 360.551,A -85,B 0,C 180,E1 -26619.599,E2 -26619.599} C_VEL
LIN {X 0,Y 101.193,Z 360.504,A -85,B 0,C 180,E1 -26627.973,E2 -26627.973} C_VEL
LIN {X 0,Y 101.273,Z 360.49,A -85,B 0,C 180,E1 -26632.021,E2 -26632.021} C_VEL
LIN {X 0,Y 101.865,Z 360.418,A -85,B 0,C 180,E1 -26639.999,E2 -26639.999} C_VEL
LIN {X 0,Y 101.273,Z 360.493,A -85,B 0,C 180,E1 -26647.977,E2 -26647.977} C_VEL
LIN {X 0,Y 101.123,Z 360.512,A -85,B 0,C 180,E1 -26653.363,E2 -26653.363} C_VEL
LIN {X 0,Y 100.812,Z 360.547,A -85,B 0,C 180,E1 -26660.399,E2 -26660.399} C_VEL
LIN {X 0,Y 100.77,Z 360.556,A -85,B 0,C 180,E1 -26664.962,E2 -26664.962} C_VEL
LIN {X 0,Y 101.12,Z 360.514,A -85,B 0,C 180,E1 -26673.779,E2 -26673.779} C_VEL
LIN {X 0,Y 101.756,Z 360.668,A -85,B 0,C 180,E1 -26678.909,E2 -26678.909} C_VEL
LIN {X 0,Y 103.212,Z 365.169,A -85,B 0,C 180,E1 -26685.203,E2 -26685.203} C_VEL
LIN {X 0,Y 103.826,Z 367.306,A -85,B 0,C 180,E1 -26688.123,E2 -26688.123} C_VEL
LIN {X 0,Y 103.252,Z 369.647,A -85,B 0,C 180,E1 -26691.14,E2 -26691.14} C_VEL
LIN {X 0,Y 102.654,Z 375.077,A -85,B 0,C 180,E1 -26692.255,E2 -26692.255} C_VEL
LIN {X 0,Y 101.929,Z 390.37,A -85,B 0,C 180,E1 -26695.457,E2 -26695.457} C_VEL
LIN {X 0,Y 102.081,Z 405.526,A -85,B 0,C 180,E1 -26699.49,E2 -26699.49} C_VEL
LIN {X 0,Y 102.995,Z 420.524,A -85,B 0,C 180,E1 -26704.365,E2 -26704.365} C_VEL
LIN {X 0,Y 104.419,Z 433.612,A -85,B 0,C 180,E1 -26709.415,E2 -26709.415} C_VEL
LIN {X 0,Y 105.776,Z 441.959,A -85,B 0,C 180,E1 -26713.105,E2 -26713.105} C_VEL
LIN {X 0,Y 105.389,Z 451.283,A -85,B 0,C 180,E1 -26718.463,E2 -26718.463} C_VEL
LIN {X 0,Y 105.891,Z 460.203,A -85,B 0,C 180,E1 -26724.587,E2 -26724.587} C_VEL
LIN {X 0,Y 107.45,Z 467.884,A -85,B 0,C 180,E1 -26730.94,E2 -26730.94} C_VEL
LIN {X 0,Y 107.64,Z 468.851,A -85,B 0,C 180,E1 -26731.874,E2 -26731.874} C_VEL
LIN {X 0,Y 107.534,Z 470.318,A -85,B 0,C 180,E1 -26733.751,E2 -26733.751} C_VEL
LIN {X 0,Y 105.285,Z 473.994,A -85,B 0,C 180,E1 -26741.555,E2 -26741.555} C_VEL
LIN {X 0,Y 105.29,Z 476.991,A -85,B 0,C 180,E1 -26750.856,E2 -26750.856} C_VEL
LIN {X 0,Y 109.202,Z 479.193,A -85,B 0,C 180,E1 -26760.992,E2 -26760.992} C_VEL
LIN {X 0,Y 114.604,Z 480.125,A -85,B 0,C 180,E1 -26767.828,E2 -26767.828} C_VEL
LIN {X 0,Y 126.059,Z 480.419,A -85,B 0,C 180,E1 -26776.454,E2 -26776.454} C_VEL
LIN {X 0,Y 130.589,Z 480.221,A -85,B 0,C 180,E1 -26778.894,E2 -26778.894} C_VEL
LIN {X 0,Y 132.546,Z 479.795,A -85,B 0,C 180,E1 -26780.486,E2 -26780.486} C_VEL
LIN {X 0,Y 121.644,Z 474.128,A -85,B 0,C 180,E1 -26786.712,E2 -26786.712} C_VEL
LIN {X 0,Y 112.655,Z 467.004,A -85,B 0,C 180,E1 -26794.108,E2 -26794.108} C_VEL
LIN {X 0,Y 107.14,Z 460.14,A -85,B 0,C 180,E1 -26800.855,E2 -26800.855} C_VEL
LIN {X 0,Y 103.146,Z 451.025,A -85,B 0,C 180,E1 -26809.201,E2 -26809.201} C_VEL
LIN {X 0,Y 101.491,Z 441.455,A -85,B 0,C 180,E1 -26817.024,E2 -26817.024} C_VEL
LIN {X 0,Y 101.075,Z 430.008,A -85,B 0,C 180,E1 -26824.987,E2 -26824.987} C_VEL
LIN {X 0,Y 101.955,Z 419.966,A -85,B 0,C 180,E1 -26830.928,E2 -26830.928} C_VEL
LIN {X 0,Y 103.583,Z 407.933,A -85,B 0,C 180,E1 -26836.921,E2 -26836.921} C_VEL
LIN {X 0,Y 105.785,Z 394.242,A -85,B 0,C 180,E1 -26842.459,E2 -26842.459} C_VEL
LIN {X 0,Y 107.179,Z 386.183,A -85,B 0,C 180,E1 -26845.229,E2 -26845.229} C_VEL
LIN {X 0,Y 103.819,Z 373.119,A -85,B 0,C 180,E1 -26849.233,E2 -26849.233} C_VEL
LIN {X 0,Y 102.709,Z 370.103,A -85,B 0,C 180,E1 -26850.37,E2 -26850.37} C_VEL
LIN {X 0,Y 100.37,Z 366.555,A -85,B 0,C 180,E1 -26852.558,E2 -26852.558} C_VEL
LIN {X 0,Y 97.803,Z 364.069,A -85,B 0,C 180,E1 -26855.206,E2 -26855.206} C_VEL
LIN {X 0,Y 95.453,Z 362.45,A -85,B 0,C 180,E1 -26858.317,E2 -26858.317} C_VEL
LIN {X 0,Y 93.584,Z 361.495,A -85,B 0,C 180,E1 -26862.955,E2 -26862.955} C_VEL
LIN {X 0,Y 93.469,Z 361.456,A -85,B 0,C 180,E1 -26864.169,E2 -26864.169} C_VEL
LIN {X 0,Y 93.552,Z 361.457,A -85,B 0,C 180,E1 -26868.7,E2 -26868.7} C_VEL
LIN {X 0,Y 93.603,Z 361.447,A -85,B 0,C 180,E1 -26875.684,E2 -26875.684} C_VEL
LIN {X 0,Y 93.674,Z 361.438,A -85,B 0,C 180,E1 -26884.203,E2 -26884.203} C_VEL
LIN {X 0,Y 93.7,Z 361.437,A -85,B 0,C 180,E1 -26887.97,E2 -26887.97} C_VEL
LIN {X 0,Y 94.103,Z 361.386,A -85,B 0,C 180,E1 -26897.049,E2 -26897.049} C_VEL
LIN {X 0,Y 94.216,Z 361.371,A -85,B 0,C 180,E1 -26901.416,E2 -26901.416} C_VEL
LIN {X 0,Y 94.801,Z 361.298,A -85,B 0,C 180,E1 -26909.996,E2 -26909.996} C_VEL
LIN {X 0,Y 94.214,Z 361.372,A -85,B 0,C 180,E1 -26918.576,E2 -26918.576} C_VEL
LIN {X 0,Y 94.049,Z 361.389,A -85,B 0,C 180,E1 -26923.717,E2 -26923.717} C_VEL
LIN {X 0,Y 93.696,Z 361.434,A -85,B 0,C 180,E1 -26932.023,E2 -26932.023} C_VEL
LIN {X 0,Y 93.621,Z 361.447,A -85,B 0,C 180,E1 -26936.766,E2 -26936.766} C_VEL
LIN {X 0,Y 93.591,Z 361.45,A -85,B 0,C 180,E1 -26944.305,E2 -26944.305} C_VEL
LIN {X 0,Y 93.532,Z 361.456,A -85,B 0,C 180,E1 -26952.547,E2 -26952.547} C_VEL
LIN {X 0,Y 93.535,Z 361.452,A -85,B 0,C 180,E1 -26958.703,E2 -26958.703} C_VEL
LIN {X 0,Y 93.59,Z 361.449,A -85,B 0,C 180,E1 -26965.685,E2 -26965.685} C_VEL
LIN {X 0,Y 93.664,Z 361.44,A -85,B 0,C 180,E1 -26974.202,E2 -26974.202} C_VEL
LIN {X 0,Y 93.69,Z 361.436,A -85,B 0,C 180,E1 -26977.97,E2 -26977.97} C_VEL
LIN {X 0,Y 94.093,Z 361.387,A -85,B 0,C 180,E1 -26987.05,E2 -26987.05} C_VEL
LIN {X 0,Y 94.205,Z 361.372,A -85,B 0,C 180,E1 -26991.418,E2 -26991.418} C_VEL
LIN {X 0,Y 94.791,Z 361.299,A -85,B 0,C 180,E1 -26999.999,E2 -26999.999} C_VEL
LIN {X 0,Y 94.205,Z 361.372,A -85,B 0,C 180,E1 -27008.58,E2 -27008.58} C_VEL
LIN {X 0,Y 94.04,Z 361.395,A -85,B 0,C 180,E1 -27013.721,E2 -27013.721} C_VEL
LIN {X 0,Y 93.688,Z 361.439,A -85,B 0,C 180,E1 -27022.028,E2 -27022.028} C_VEL
LIN {X 0,Y 93.686,Z 361.433,A -85,B 0,C 180,E1 -27026.749,E2 -27026.749} C_VEL
LIN {X 0,Y 94.142,Z 361.382,A -85,B 0,C 180,E1 -27034.804,E2 -27034.804} C_VEL
LIN {X 0,Y 94.835,Z 361.408,A -85,B 0,C 180,E1 -27040.075,E2 -27040.075} C_VEL
LIN {X 0,Y 96.384,Z 365.9,A -85,B 0,C 180,E1 -27046.815,E2 -27046.815} C_VEL
LIN {X 0,Y 96.594,Z 367.432,A -85,B 0,C 180,E1 -27049.099,E2 -27049.099} C_VEL
LIN {X 0,Y 96.261,Z 368.596,A -85,B 0,C 180,E1 -27050.639,E2 -27050.639} C_VEL
LIN {X 0,Y 94.986,Z 386.081,A -85,B 0,C 180,E1 -27054.476,E2 -27054.476} C_VEL
LIN {X 0,Y 94.923,Z 401.735,A -85,B 0,C 180,E1 -27058.788,E2 -27058.788} C_VEL
LIN {X 0,Y 95.636,Z 415.607,A -85,B 0,C 180,E1 -27063.437,E2 -27063.437} C_VEL
LIN {X 0,Y 97.076,Z 429.056,A -85,B 0,C 180,E1 -27068.782,E2 -27068.782} C_VEL
LIN {X 0,Y 99.015,Z 440.509,A -85,B 0,C 180,E1 -27074.039,E2 -27074.039} C_VEL
LIN {X 0,Y 98.834,Z 449.795,A -85,B 0,C 180,E1 -27079.764,E2 -27079.764} C_VEL
LIN {X 0,Y 99.516,Z 458.244,A -85,B 0,C 180,E1 -27085.954,E2 -27085.954} C_VEL
LIN {X 0,Y 101.151,Z 465.233,A -85,B 0,C 180,E1 -27091.994,E2 -27091.994} C_VEL
LIN {X 0,Y 101.262,Z 466.959,A -85,B 0,C 180,E1 -27093.983,E2 -27093.983} C_VEL
LIN {X 0,Y 99.022,Z 470.763,A -85,B 0,C 180,E1 -27102.297,E2 -27102.297} C_VEL
LIN {X 0,Y 99.452,Z 474.255,A -85,B 0,C 180,E1 -27113.269,E2 -27113.269} C_VEL
LIN {X 0,Y 103.55,Z 476.45,A -85,B 0,C 180,E1 -27122.89,E2 -27122.89} C_VEL
LIN {X 0,Y 109.391,Z 477.547,A -85,B 0,C 180,E1 -27129.98,E2 -27129.98} C_VEL
LIN {X 0,Y 121.47,Z 478.201,A -85,B 0,C 180,E1 -27138.781,E2 -27138.781} C_VEL
LIN {X 0,Y 122.625,Z 478.187,A -85,B 0,C 180,E1 -27139.42,E2 -27139.42} C_VEL
LIN {X 0,Y 123.219,Z 477.858,A -85,B 0,C 180,E1 -27140.403,E2 -27140.403} C_VEL
LIN {X 0,Y 111.767,Z 470.805,A -85,B 0,C 180,E1 -27147.692,E2 -27147.692} C_VEL
LIN {X 0,Y 103.234,Z 462.602,A -85,B 0,C 180,E1 -27155.892,E2 -27155.892} C_VEL
LIN {X 0,Y 97.92,Z 453.761,A -85,B 0,C 180,E1 -27164.387,E2 -27164.387} C_VEL
LIN {X 0,Y 95.038,Z 443.269,A -85,B 0,C 180,E1 -27173.632,E2 -27173.632} C_VEL
LIN {X 0,Y 94.221,Z 435.09,A -85,B 0,C 180,E1 -27180.001,E2 -27180.001} C_VEL
LIN {X 0,Y 94.682,Z 422.339,A -85,B 0,C 180,E1 -27188.539,E2 -27188.539} C_VEL
LIN {X 0,Y 95.929,Z 410.953,A -85,B 0,C 180,E1 -27194.859,E2 -27194.859} C_VEL
LIN {X 0,Y 97.857,Z 398.896,A -85,B 0,C 180,E1 -27200.418,E2 -27200.418} C_VEL
LIN {X 0,Y 99.919,Z 386.13,A -85,B 0,C 180,E1 -27205.272,E2 -27205.272} C_VEL
LIN {X 0,Y 96.299,Z 372.247,A -85,B 0,C 180,E1 -27209.731,E2 -27209.731} C_VEL
LIN {X 0,Y 94.001,Z 362,A -85,B 0,C 180,E1 -27212.822,E2 -27212.822} C_VEL
LIN {X 0,Y 93.835,Z 361.46,A -85,B 0,C 180,E1 -27213.528,E2 -27213.528} C_VEL
LIN {X 0,Y 93.544,Z 361.456,A -85,B 0,C 180,E1 -27222.547,E2 -27222.547} C_VEL
LIN {X 0,Y 93.469,Z 361.456,A -85,B 0,C 180,E1 -27224.169,E2 -27224.169} C_VEL
LIN {X 0,Y 92.774,Z 361.552,A -85,B 0,C 180,E1 -27227.771,E2 -27227.771} C_VEL
LIN {X 0,Y 91.248,Z 361.742,A -85,B 0,C 180,E1 -27231.347,E2 -27231.347} C_VEL
LIN {X 0,Y 86.892,Z 362.282,A -85,B 0,C 180,E1 -27241.376,E2 -27241.376} C_VEL
LIN {X 0,Y 86.568,Z 362.32,A -85,B 0,C 180,E1 -27244.047,E2 -27244.047} C_VEL
LIN {X 0,Y 86.653,Z 362.308,A -85,B 0,C 180,E1 -27251.065,E2 -27251.065} C_VEL
LIN {X 0,Y 86.974,Z 362.276,A -85,B 0,C 180,E1 -27255.967,E2 -27255.967} C_VEL
LIN {X 0,Y 87.122,Z 362.253,A -85,B 0,C 180,E1 -27260.711,E2 -27260.711} C_VEL
LIN {X 0,Y 87.729,Z 362.179,A -85,B 0,C 180,E1 -27269.996,E2 -27269.996} C_VEL
LIN {X 0,Y 87.12,Z 362.256,A -85,B 0,C 180,E1 -27279.28,E2 -27279.28} C_VEL
LIN {X 0,Y 86.952,Z 362.272,A -85,B 0,C 180,E1 -27284.083,E2 -27284.083} C_VEL
LIN {X 0,Y 86.666,Z 362.314,A -85,B 0,C 180,E1 -27288.923,E2 -27288.923} C_VEL
LIN {X 0,Y 86.583,Z 362.324,A -85,B 0,C 180,E1 -27296.76,E2 -27296.76} C_VEL
LIN {X 0,Y 86.509,Z 362.334,A -85,B 0,C 180,E1 -27305.666,E2 -27305.666} C_VEL
LIN {X 0,Y 86.474,Z 362.336,A -85,B 0,C 180,E1 -27312.99,E2 -27312.99} C_VEL
LIN {X 0,Y 86.456,Z 362.333,A -85,B 0,C 180,E1 -27319.433,E2 -27319.433} C_VEL
LIN {X 0,Y 86.533,Z 362.328,A -85,B 0,C 180,E1 -27325.351,E2 -27325.351} C_VEL
LIN {X 0,Y 86.581,Z 362.324,A -85,B 0,C 180,E1 -27333.23,E2 -27333.23} C_VEL
LIN {X 0,Y 86.66,Z 362.315,A -85,B 0,C 180,E1 -27341.07,E2 -27341.07} C_VEL
LIN {X 0,Y 86.964,Z 362.272,A -85,B 0,C 180,E1 -27345.968,E2 -27345.968} C_VEL
LIN {X 0,Y 87.112,Z 362.257,A -85,B 0,C 180,E1 -27350.713,E2 -27350.713} C_VEL
LIN {X 0,Y 87.719,Z 362.18,A -85,B 0,C 180,E1 -27359.999,E2 -27359.999} C_VEL
LIN {X 0,Y 87.111,Z 362.253,A -85,B 0,C 180,E1 -27369.284,E2 -27369.284} C_VEL
LIN {X 0,Y 86.944,Z 362.28,A -85,B 0,C 180,E1 -27374.087,E2 -27374.087} C_VEL
LIN {X 0,Y 86.599,Z 362.323,A -85,B 0,C 180,E1 -27383.939,E2 -27383.939} C_VEL
LIN {X 0,Y 86.637,Z 362.314,A -85,B 0,C 180,E1 -27389.124,E2 -27389.124} C_VEL
LIN {X 0,Y 87.247,Z 362.239,A -85,B 0,C 180,E1 -27396.346,E2 -27396.346} C_VEL
LIN {X 0,Y 88.081,Z 362.325,A -85,B 0,C 180,E1 -27401.93,E2 -27401.93} C_VEL
LIN {X 0,Y 89.408,Z 366.149,A -85,B 0,C 180,E1 -27408.081,E2 -27408.081} C_VEL
LIN {X 0,Y 89.312,Z 367.539,A -85,B 0,C 180,E1 -27410.078,E2 -27410.078} C_VEL
LIN {X 0,Y 88.657,Z 372.896,A -85,B 0,C 180,E1 -27411.382,E2 -27411.382} C_VEL
LIN {X 0,Y 87.791,Z 389.052,A -85,B 0,C 180,E1 -27415.379,E2 -27415.379} C_VEL
LIN {X 0,Y 87.976,Z 404.584,A -85,B 0,C 180,E1 -27420.303,E2 -27420.303} C_VEL
LIN {X 0,Y 89.018,Z 418.294,A -85,B 0,C 180,E1 -27425.518,E2 -27425.518} C_VEL
LIN {X 0,Y 90.623,Z 430.855,A -85,B 0,C 180,E1 -27431.097,E2 -27431.097} C_VEL
LIN {X 0,Y 92.341,Z 439.897,A -85,B 0,C 180,E1 -27435.683,E2 -27435.683} C_VEL
LIN {X 0,Y 92.497,Z 450.196,A -85,B 0,C 180,E1 -27442.692,E2 -27442.692} C_VEL
LIN {X 0,Y 93.888,Z 459.111,A -85,B 0,C 180,E1 -27450.004,E2 -27450.004} C_VEL
LIN {X 0,Y 94.561,Z 461.4,A -85,B 0,C 180,E1 -27452.134,E2 -27452.134} C_VEL
LIN {X 0,Y 94.995,Z 463.382,A -85,B 0,C 180,E1 -27454.247,E2 -27454.247} C_VEL
LIN {X 0,Y 92.837,Z 467.419,A -85,B 0,C 180,E1 -27463.131,E2 -27463.131} C_VEL
LIN {X 0,Y 94.059,Z 471.605,A -85,B 0,C 180,E1 -27476.64,E2 -27476.64} C_VEL
LIN {X 0,Y 100.991,Z 474.254,A -85,B 0,C 180,E1 -27488.783,E2 -27488.783} C_VEL
LIN {X 0,Y 112.515,Z 475.625,A -85,B 0,C 180,E1 -27498.556,E2 -27498.556} C_VEL
LIN {X 0,Y 113.671,Z 475.161,A -85,B 0,C 180,E1 -27500.453,E2 -27500.453} C_VEL
LIN {X 0,Y 103.826,Z 468.305,A -85,B 0,C 180,E1 -27507.214,E2 -27507.214} C_VEL
LIN {X 0,Y 95.438,Z 459.328,A -85,B 0,C 180,E1 -27516.109,E2 -27516.109} C_VEL
LIN {X 0,Y 90.359,Z 449.739,A -85,B 0,C 180,E1 -27525.359,E2 -27525.359} C_VEL
LIN {X 0,Y 87.876,Z 438.402,A -85,B 0,C 180,E1 -27535.414,E2 -27535.414} C_VEL
LIN {X 0,Y 87.339,Z 426.166,A -85,B 0,C 180,E1 -27544.617,E2 -27544.617} C_VEL
LIN {X 0,Y 88.256,Z 415.439,A -85,B 0,C 180,E1 -27551.484,E2 -27551.484} C_VEL
LIN {X 0,Y 90.051,Z 402.79,A -85,B 0,C 180,E1 -27558.192,E2 -27558.192} C_VEL
LIN {X 0,Y 92.182,Z 389.835,A -85,B 0,C 180,E1 -27563.801,E2 -27563.801} C_VEL
LIN {X 0,Y 92.749,Z 386.582,A -85,B 0,C 180,E1 -27565.05,E2 -27565.05} C_VEL
LIN {X 0,Y 89.121,Z 372.586,A -85,B 0,C 180,E1 -27569.829,E2 -27569.829} C_VEL
LIN {X 0,Y 86.937,Z 362.941,A -85,B 0,C 180,E1 -27572.948,E2 -27572.948} C_VEL
LIN {X 0,Y 86.725,Z 362.33,A -85,B 0,C 180,E1 -27573.955,E2 -27573.955} C_VEL
LIN {X 0,Y 86.486,Z 362.334,A -85,B 0,C 180,E1 -27582.995,E2 -27582.995} C_VEL
LIN {X 0,Y 86.472,Z 362.338,A -85,B 0,C 180,E1 -27589.438,E2 -27589.438} C_VEL
LIN {X 0,Y 86.547,Z 362.326,A -85,B 0,C 180,E1 -27595.354,E2 -27595.354} C_VEL
LIN {X 0,Y 86.568,Z 362.32,A -85,B 0,C 180,E1 -27604.047,E2 -27604.047} C_VEL
LIN {X 0,Y 85.893,Z 362.412,A -85,B 0,C 180,E1 -27607.938,E2 -27607.938} C_VEL
LIN {X 0,Y 84.393,Z 362.607,A -85,B 0,C 180,E1 -27611.81,E2 -27611.81} C_VEL
LIN {X 0,Y 80.333,Z 363.112,A -85,B 0,C 180,E1 -27622.721,E2 -27622.721} C_VEL
LIN {X 0,Y 80.18,Z 363.117,A -85,B 0,C 180,E1 -27625.615,E2 -27625.615} C_VEL
LIN {X 0,Y 80.657,Z 363.06,A -85,B 0,C 180,E1 -27629.995,E2 -27629.995} C_VEL
LIN {X 0,Y 80.003,Z 363.145,A -85,B 0,C 180,E1 -27640.114,E2 -27640.114} C_VEL
LIN {X 0,Y 79.767,Z 363.165,A -85,B 0,C 180,E1 -27645.322,E2 -27645.322} C_VEL
LIN {X 0,Y 79.525,Z 363.203,A -85,B 0,C 180,E1 -27650.696,E2 -27650.696} C_VEL
LIN {X 0,Y 79.481,Z 363.21,A -85,B 0,C 180,E1 -27657.839,E2 -27657.839} C_VEL
LIN {X 0,Y 79.379,Z 363.213,A -85,B 0,C 180,E1 -27662.083,E2 -27662.083} C_VEL
LIN {X 0,Y 79.366,Z 363.222,A -85,B 0,C 180,E1 -27668.3,E2 -27668.3} C_VEL
LIN {X 0,Y 79.383,Z 363.222,A -85,B 0,C 180,E1 -27675.087,E2 -27675.087} C_VEL
LIN {X 0,Y 79.386,Z 363.221,A -85,B 0,C 180,E1 -27682.814,E2 -27682.814} C_VEL
LIN {X 0,Y 79.377,Z 363.214,A -85,B 0,C 180,E1 -27687.909,E2 -27687.909} C_VEL
LIN {X 0,Y 79.521,Z 363.203,A -85,B 0,C 180,E1 -27693.774,E2 -27693.774} C_VEL
LIN {X 0,Y 79.519,Z 363.204,A -85,B 0,C 180,E1 -27699.295,E2 -27699.295} C_VEL
LIN {X 0,Y 79.836,Z 363.158,A -85,B 0,C 180,E1 -27705.523,E2 -27705.523} C_VEL
LIN {X 0,Y 79.994,Z 363.145,A -85,B 0,C 180,E1 -27709.878,E2 -27709.878} C_VEL
LIN {X 0,Y 80.647,Z 363.06,A -85,B 0,C 180,E1 -27719.999,E2 -27719.999} C_VEL
LIN {X 0,Y 79.994,Z 363.137,A -85,B 0,C 180,E1 -27730.119,E2 -27730.119} C_VEL
LIN {X 0,Y 79.756,Z 363.175,A -85,B 0,C 180,E1 -27735.327,E2 -27735.327} C_VEL
LIN {X 0,Y 79.515,Z 363.2,A -85,B 0,C 180,E1 -27740.703,E2 -27740.703} C_VEL
LIN {X 0,Y 79.581,Z 363.189,A -85,B 0,C 180,E1 -27747.988,E2 -27747.988} C_VEL
LIN {X 0,Y 80.393,Z 363.094,A -85,B 0,C 180,E1 -27758.122,E2 -27758.122} C_VEL
LIN {X 0,Y 81.39,Z 363.218,A -85,B 0,C 180,E1 -27764.114,E2 -27764.114} C_VEL
LIN {X 0,Y 82.333,Z 366.136,A -85,B 0,C 180,E1 -27769.088,E2 -27769.088} C_VEL
LIN {X 0,Y 82.304,Z 366.663,A -85,B 0,C 180,E1 -27769.673,E2 -27769.673} C_VEL
LIN {X 0,Y 80.867,Z 383.838,A -85,B 0,C 180,E1 -27774.088,E2 -27774.088} C_VEL
LIN {X 0,Y 80.783,Z 399.133,A -85,B 0,C 180,E1 -27779.073,E2 -27779.073} C_VEL
LIN {X 0,Y 81.614,Z 412.96,A -85,B 0,C 180,E1 -27784.502,E2 -27784.502} C_VEL
LIN {X 0,Y 83.413,Z 426.868,A -85,B 0,C 180,E1 -27790.949,E2 -27790.949} C_VEL
LIN {X 0,Y 85.732,Z 438.389,A -85,B 0,C 180,E1 -27797.097,E2 -27797.097} C_VEL
LIN {X 0,Y 86.197,Z 448.495,A -85,B 0,C 180,E1 -27804.508,E2 -27804.508} C_VEL
LIN {X 0,Y 87.966,Z 457.355,A -85,B 0,C 180,E1 -27812.294,E2 -27812.294} C_VEL
LIN {X 0,Y 88.636,Z 459.567,A -85,B 0,C 180,E1 -27814.552,E2 -27814.552} C_VEL
LIN {X 0,Y 88.225,Z 460.955,A -85,B 0,C 180,E1 -27816.867,E2 -27816.867} C_VEL
LIN {X 0,Y 86.58,Z 465.579,A -85,B 0,C 180,E1 -27828.951,E2 -27828.951} C_VEL
LIN {X 0,Y 90.297,Z 469.465,A -85,B 0,C 180,E1 -27843.017,E2 -27843.017} C_VEL
LIN {X 0,Y 99.637,Z 471.971,A -85,B 0,C 180,E1 -27854.863,E2 -27854.863} C_VEL
LIN {X 0,Y 104.71,Z 472.626,A -85,B 0,C 180,E1 -27858.886,E2 -27858.886} C_VEL
LIN {X 0,Y 104.2,Z 471.716,A -85,B 0,C 180,E1 -27860.553,E2 -27860.553} C_VEL
LIN {X 0,Y 94.197,Z 463.539,A -85,B 0,C 180,E1 -27868.517,E2 -27868.517} C_VEL
LIN {X 0,Y 86.38,Z 453.445,A -85,B 0,C 180,E1 -27878.524,E2 -27878.524} C_VEL
LIN {X 0,Y 82.568,Z 443.983,A -85,B 0,C 180,E1 -27887.715,E2 -27887.715} C_VEL
LIN {X 0,Y 80.868,Z 434.354,A -85,B 0,C 180,E1 -27896.264,E2 -27896.264} C_VEL
LIN {X 0,Y 80.58,Z 423.075,A -85,B 0,C 180,E1 -27905.005,E2 -27905.005} C_VEL
LIN {X 0,Y 81.356,Z 413.78,A -85,B 0,C 180,E1 -27911.209,E2 -27911.209} C_VEL
LIN {X 0,Y 83.355,Z 399.68,A -85,B 0,C 180,E1 -27919.071,E2 -27919.071} C_VEL
LIN {X 0,Y 85.327,Z 387.992,A -85,B 0,C 180,E1 -27924.321,E2 -27924.321} C_VEL
LIN {X 0,Y 85.365,Z 386.029,A -85,B 0,C 180,E1 -27925.084,E2 -27925.084} C_VEL
LIN {X 0,Y 81.512,Z 371.29,A -85,B 0,C 180,E1 -27930.427,E2 -27930.427} C_VEL
LIN {X 0,Y 79.851,Z 363.731,A -85,B 0,C 180,E1 -27933.1,E2 -27933.1} C_VEL
LIN {X 0,Y 79.638,Z 363.207,A -85,B 0,C 180,E1 -27934.237,E2 -27934.237} C_VEL
LIN {X 0,Y 79.437,Z 363.21,A -85,B 0,C 180,E1 -27938.268,E2 -27938.268} C_VEL
LIN {X 0,Y 79.416,Z 363.209,A -85,B 0,C 180,E1 -27945.072,E2 -27945.072} C_VEL
LIN {X 0,Y 79.399,Z 363.212,A -85,B 0,C 180,E1 -27952.812,E2 -27952.812} C_VEL
LIN {X 0,Y 79.389,Z 363.221,A -85,B 0,C 180,E1 -27957.911,E2 -27957.911} C_VEL
LIN {X 0,Y 79.527,Z 363.198,A -85,B 0,C 180,E1 -27963.82,E2 -27963.82} C_VEL
LIN {X 0,Y 79.52,Z 363.199,A -85,B 0,C 180,E1 -27969.292,E2 -27969.292} C_VEL
LIN {X 0,Y 79.846,Z 363.164,A -85,B 0,C 180,E1 -27975.522,E2 -27975.522} C_VEL
LIN {X 0,Y 80.005,Z 363.136,A -85,B 0,C 180,E1 -27979.877,E2 -27979.877} C_VEL
LIN {X 0,Y 80.18,Z 363.117,A -85,B 0,C 180,E1 -27985.615,E2 -27985.615} C_VEL
LIN {X 0,Y 79.963,Z 363.142,A -85,B 0,C 180,E1 -27988.412,E2 -27988.412} C_VEL
LIN {X 0,Y 78.624,Z 363.316,A -85,B 0,C 180,E1 -27992.571,E2 -27992.571} C_VEL
LIN {X 0,Y 76.646,Z 363.554,A -85,B 0,C 180,E1 -27996.729,E2 -27996.729} C_VEL
LIN {X 0,Y 72.908,Z 364.021,A -85,B 0,C 180,E1 -28005.788,E2 -28005.788} C_VEL
LIN {X 0,Y 72.43,Z 364.071,A -85,B 0,C 180,E1 -28009.017,E2 -28009.017} C_VEL
LIN {X 0,Y 72.4,Z 364.084,A -85,B 0,C 180,E1 -28012.842,E2 -28012.842} C_VEL
LIN {X 0,Y 72.376,Z 364.093,A -85,B 0,C 180,E1 -28019.077,E2 -28019.077} C_VEL
LIN {X 0,Y 72.294,Z 364.105,A -85,B 0,C 180,E1 -28025.675,E2 -28025.675} C_VEL
LIN {X 0,Y 72.244,Z 364.108,A -85,B 0,C 180,E1 -28032.912,E2 -28032.912} C_VEL
LIN {X 0,Y 72.292,Z 364.1,A -85,B 0,C 180,E1 -28041.045,E2 -28041.045} C_VEL
LIN {X 0,Y 72.293,Z 364.105,A -85,B 0,C 180,E1 -28044.316,E2 -28044.316} C_VEL
LIN {X 0,Y 72.37,Z 364.095,A -85,B 0,C 180,E1 -28050.949,E2 -28050.949} C_VEL
LIN {X 0,Y 72.395,Z 364.084,A -85,B 0,C 180,E1 -28057.149,E2 -28057.149} C_VEL
LIN {X 0,Y 72.752,Z 364.039,A -85,B 0,C 180,E1 -28065,E2 -28065} C_VEL
LIN {X 0,Y 72.879,Z 364.032,A -85,B 0,C 180,E1 -28068.878,E2 -28068.878} C_VEL
LIN {X 0,Y 73.574,Z 363.941,A -85,B 0,C 180,E1 -28079.999,E2 -28079.999} C_VEL
LIN {X 0,Y 72.878,Z 364.024,A -85,B 0,C 180,E1 -28091.119,E2 -28091.119} C_VEL
LIN {X 0,Y 72.578,Z 364.066,A -85,B 0,C 180,E1 -28096.887,E2 -28096.887} C_VEL
LIN {X 0,Y 72.409,Z 364.09,A -85,B 0,C 180,E1 -28102.843,E2 -28102.843} C_VEL
LIN {X 0,Y 72.534,Z 364.07,A -85,B 0,C 180,E1 -28109.316,E2 -28109.316} C_VEL
LIN {X 0,Y 73.547,Z 363.946,A -85,B 0,C 180,E1 -28120.149,E2 -28120.149} C_VEL
LIN {X 0,Y 74.725,Z 363.92,A -85,B 0,C 180,E1 -28126.303,E2 -28126.303} C_VEL
LIN {X 0,Y 75.205,Z 365.68,A -85,B 0,C 180,E1 -28129.151,E2 -28129.151} C_VEL
LIN {X 0,Y 73.773,Z 383.76,A -85,B 0,C 180,E1 -28134.31,E2 -28134.31} C_VEL
LIN {X 0,Y 73.771,Z 399.296,A -85,B 0,C 180,E1 -28139.961,E2 -28139.961} C_VEL
LIN {X 0,Y 74.931,Z 414.135,A -85,B 0,C 180,E1 -28146.513,E2 -28146.513} C_VEL
LIN {X 0,Y 77.055,Z 427.625,A -85,B 0,C 180,E1 -28153.445,E2 -28153.445} C_VEL
LIN {X 0,Y 79.215,Z 436.774,A -85,B 0,C 180,E1 -28158.748,E2 -28158.748} C_VEL
LIN {X 0,Y 79.952,Z 446.24,A -85,B 0,C 180,E1 -28166.225,E2 -28166.225} C_VEL
LIN {X 0,Y 82.225,Z 455.491,A -85,B 0,C 180,E1 -28174.908,E2 -28174.908} C_VEL
LIN {X 0,Y 82.214,Z 457.193,A -85,B 0,C 180,E1 -28177.372,E2 -28177.372} C_VEL
LIN {X 0,Y 80.713,Z 462.027,A -85,B 0,C 180,E1 -28190.388,E2 -28190.388} C_VEL
LIN {X 0,Y 85.018,Z 466.156,A -85,B 0,C 180,E1 -28205.361,E2 -28205.361} C_VEL
LIN {X 0,Y 95.135,Z 468.94,A -85,B 0,C 180,E1 -28217.629,E2 -28217.629} C_VEL
LIN {X 0,Y 96.86,Z 469.137,A -85,B 0,C 180,E1 -28219.231,E2 -28219.231} C_VEL
LIN {X 0,Y 86.446,Z 459.974,A -85,B 0,C 180,E1 -28228.101,E2 -28228.101} C_VEL
LIN {X 0,Y 79.418,Z 450.231,A -85,B 0,C 180,E1 -28237.909,E2 -28237.909} C_VEL
LIN {X 0,Y 75.287,Z 438.778,A -85,B 0,C 180,E1 -28249.241,E2 -28249.241} C_VEL
LIN {X 0,Y 73.923,Z 429.879,A -85,B 0,C 180,E1 -28257.277,E2 -28257.277} C_VEL
LIN {X 0,Y 74.053,Z 417.851,A -85,B 0,C 180,E1 -28266.815,E2 -28266.815} C_VEL
LIN {X 0,Y 75.42,Z 404.448,A -85,B 0,C 180,E1 -28275.541,E2 -28275.541} C_VEL
LIN {X 0,Y 77.591,Z 391.137,A -85,B 0,C 180,E1 -28282.536,E2 -28282.536} C_VEL
LIN {X 0,Y 78.269,Z 386.951,A -85,B 0,C 180,E1 -28284.43,E2 -28284.43} C_VEL
LIN {X 0,Y 74.768,Z 373.468,A -85,B 0,C 180,E1 -28289.73,E2 -28289.73} C_VEL
LIN {X 0,Y 72.883,Z 365.034,A -85,B 0,C 180,E1 -28292.865,E2 -28292.865} C_VEL
LIN {X 0,Y 72.613,Z 364.111,A -85,B 0,C 180,E1 -28293.991,E2 -28293.991} C_VEL
LIN {X 0,Y 72.282,Z 364.103,A -85,B 0,C 180,E1 -28302.894,E2 -28302.894} C_VEL
LIN {X 0,Y 72.307,Z 364.101,A -85,B 0,C 180,E1 -28311.042,E2 -28311.042} C_VEL
LIN {X 0,Y 72.305,Z 364.095,A -85,B 0,C 180,E1 -28314.319,E2 -28314.319} C_VEL
LIN {X 0,Y 72.38,Z 364.088,A -85,B 0,C 180,E1 -28320.95,E2 -28320.95} C_VEL
LIN {X 0,Y 72.4,Z 364.091,A -85,B 0,C 180,E1 -28327.147,E2 -28327.147} C_VEL
LIN {X 0,Y 72.741,Z 364.049,A -85,B 0,C 180,E1 -28335.061,E2 -28335.061} C_VEL
LIN {X 0,Y 72.889,Z 364.022,A -85,B 0,C 180,E1 -28338.876,E2 -28338.876} C_VEL
LIN {X 0,Y 73.584,Z 363.94,A -85,B 0,C 180,E1 -28349.995,E2 -28349.995} C_VEL
LIN {X 0,Y 72.887,Z 364.031,A -85,B 0,C 180,E1 -28361.114,E2 -28361.114} C_VEL
LIN {X 0,Y 72.587,Z 364.064,A -85,B 0,C 180,E1 -28366.88,E2 -28366.88} C_VEL
LIN {X 0,Y 72.43,Z 364.071,A -85,B 0,C 180,E1 -28369.017,E2 -28369.017} C_VEL
LIN {X 0,Y 71.981,Z 364.138,A -85,B 0,C 180,E1 -28372.114,E2 -28372.114} C_VEL
LIN {X 0,Y 70.516,Z 364.325,A -85,B 0,C 180,E1 -28376.728,E2 -28376.728} C_VEL
LIN {X 0,Y 67.269,Z 364.729,A -85,B 0,C 180,E1 -28384.646,E2 -28384.646} C_VEL
LIN {X 0,Y 65.321,Z 364.965,A -85,B 0,C 180,E1 -28391.512,E2 -28391.512} C_VEL
LIN {X 0,Y 65.02,Z 364.982,A -85,B 0,C 180,E1 -28395.092,E2 -28395.092} C_VEL
LIN {X 0,Y 65.199,Z 364.98,A -85,B 0,C 180,E1 -28399.7,E2 -28399.7} C_VEL
LIN {X 0,Y 65.25,Z 364.977,A -85,B 0,C 180,E1 -28409.493,E2 -28409.493} C_VEL
LIN {X 0,Y 65.237,Z 364.978,A -85,B 0,C 180,E1 -28414.472,E2 -28414.472} C_VEL
LIN {X 0,Y 65.646,Z 364.924,A -85,B 0,C 180,E1 -28424.456,E2 -28424.456} C_VEL
LIN {X 0,Y 65.778,Z 364.915,A -85,B 0,C 180,E1 -28427.66,E2 -28427.66} C_VEL
LIN {X 0,Y 66.498,Z 364.822,A -85,B 0,C 180,E1 -28439.998,E2 -28439.998} C_VEL
LIN {X 0,Y 65.769,Z 364.913,A -85,B 0,C 180,E1 -28452.339,E2 -28452.339} C_VEL
LIN {X 0,Y 65.387,Z 364.956,A -85,B 0,C 180,E1 -28458.809,E2 -28458.809} C_VEL
LIN {X 0,Y 65.316,Z 364.97,A -85,B 0,C 180,E1 -28465.491,E2 -28465.491} C_VEL
LIN {X 0,Y 65.572,Z 364.942,A -85,B 0,C 180,E1 -28472.403,E2 -28472.403} C_VEL
LIN {X 0,Y 66.817,Z 364.783,A -85,B 0,C 180,E1 -28482.593,E2 -28482.593} C_VEL
LIN {X 0,Y 67.869,Z 364.805,A -85,B 0,C 180,E1 -28488.021,E2 -28488.021} C_VEL
LIN {X 0,Y 68.077,Z 365.826,A -85,B 0,C 180,E1 -28489.007,E2 -28489.007} C_VEL
LIN {X 0,Y 66.764,Z 382.164,A -85,B 0,C 180,E1 -28494.148,E2 -28494.148} C_VEL
LIN {X 0,Y 66.756,Z 397.833,A -85,B 0,C 180,E1 -28500.436,E2 -28500.436} C_VEL
LIN {X 0,Y 68.033,Z 412.577,A -85,B 0,C 180,E1 -28507.573,E2 -28507.573} C_VEL
LIN {X 0,Y 70.345,Z 425.888,A -85,B 0,C 180,E1 -28515.024,E2 -28515.024} C_VEL
LIN {X 0,Y 72.67,Z 434.615,A -85,B 0,C 180,E1 -28520.412,E2 -28520.412} C_VEL
LIN {X 0,Y 73.637,Z 442.854,A -85,B 0,C 180,E1 -28527.27,E2 -28527.27} C_VEL
LIN {X 0,Y 75.7,Z 451.125,A -85,B 0,C 180,E1 -28535.332,E2 -28535.332} C_VEL
LIN {X 0,Y 76.198,Z 452.351,A -85,B 0,C 180,E1 -28536.625,E2 -28536.625} C_VEL
LIN {X 0,Y 76.283,Z 453.258,A -85,B 0,C 180,E1 -28537.948,E2 -28537.948} C_VEL
LIN {X 0,Y 75.016,Z 458.291,A -85,B 0,C 180,E1 -28552.014,E2 -28552.014} C_VEL
LIN {X 0,Y 77.601,Z 461.401,A -85,B 0,C 180,E1 -28562.92,E2 -28562.92} C_VEL
LIN {X 0,Y 86.752,Z 464.825,A -85,B 0,C 180,E1 -28576.818,E2 -28576.818} C_VEL
LIN {X 0,Y 87.662,Z 465.048,A -85,B 0,C 180,E1 -28577.698,E2 -28577.698} C_VEL
LIN {X 0,Y 87.015,Z 463.972,A -85,B 0,C 180,E1 -28579.75,E2 -28579.75} C_VEL
LIN {X 0,Y 76.994,Z 453.668,A -85,B 0,C 180,E1 -28589.866,E2 -28589.866} C_VEL
LIN {X 0,Y 70.796,Z 442.819,A -85,B 0,C 180,E1 -28601.18,E2 -28601.18} C_VEL
LIN {X 0,Y 68.129,Z 433.004,A -85,B 0,C 180,E1 -28611.1,E2 -28611.1} C_VEL
LIN {X 0,Y 67.056,Z 419.66,A -85,B 0,C 180,E1 -28623.005,E2 -28623.005} C_VEL
LIN {X 0,Y 67.823,Z 408.884,A -85,B 0,C 180,E1 -28631.205,E2 -28631.205} C_VEL
LIN {X 0,Y 69.77,Z 394.908,A -85,B 0,C 180,E1 -28639.877,E2 -28639.877} C_VEL
LIN {X 0,Y 71.045,Z 387.202,A -85,B 0,C 180,E1 -28643.857,E2 -28643.857} C_VEL
LIN {X 0,Y 68.128,Z 375.859,A -85,B 0,C 180,E1 -28648.725,E2 -28648.725} C_VEL
LIN {X 0,Y 65.763,Z 365.534,A -85,B 0,C 180,E1 -28653.024,E2 -28653.024} C_VEL
LIN {X 0,Y 65.54,Z 364.973,A -85,B 0,C 180,E1 -28654.264,E2 -28654.264} C_VEL
LIN {X 0,Y 65.228,Z 364.985,A -85,B 0,C 180,E1 -28661.035,E2 -28661.035} C_VEL
LIN {X 0,Y 65.218,Z 364.986,A -85,B 0,C 180,E1 -28669.709,E2 -28669.709} C_VEL
LIN {X 0,Y 65.26,Z 364.979,A -85,B 0,C 180,E1 -28679.494,E2 -28679.494} C_VEL
LIN {X 0,Y 65.244,Z 364.979,A -85,B 0,C 180,E1 -28684.471,E2 -28684.471} C_VEL
LIN {X 0,Y 65.641,Z 364.934,A -85,B 0,C 180,E1 -28694.502,E2 -28694.502} C_VEL
LIN {X 0,Y 65.78,Z 364.91,A -85,B 0,C 180,E1 -28697.656,E2 -28697.656} C_VEL
LIN {X 0,Y 66.508,Z 364.821,A -85,B 0,C 180,E1 -28709.995,E2 -28709.995} C_VEL
LIN {X 0,Y 65.785,Z 364.914,A -85,B 0,C 180,E1 -28722.331,E2 -28722.331} C_VEL
LIN {X 0,Y 65.392,Z 364.964,A -85,B 0,C 180,E1 -28728.804,E2 -28728.804} C_VEL
LIN {X 0,Y 65.241,Z 364.979,A -85,B 0,C 180,E1 -28735.518,E2 -28735.518} C_VEL
LIN {X 0,Y 65.195,Z 364.98,A -85,B 0,C 180,E1 -28742.609,E2 -28742.609} C_VEL
LIN {X 0,Y 65.18,Z 364.982,A -85,B 0,C 180,E1 -28750.992,E2 -28750.992} C_VEL
LIN {X 0,Y 65.02,Z 364.982,A -85,B 0,C 180,E1 -28755.092,E2 -28755.092} C_VEL
LIN {X 0,Y 64.714,Z 365.04,A -85,B 0,C 180,E1 -28758.548,E2 -28758.548} C_VEL
LIN {X 0,Y 63.421,Z 365.21,A -85,B 0,C 180,E1 -28763.715,E2 -28763.715} C_VEL
LIN {X 0,Y 60.418,Z 365.584,A -85,B 0,C 180,E1 -28772.627,E2 -28772.627} C_VEL
LIN {X 0,Y 58.703,Z 365.798,A -85,B 0,C 180,E1 -28780.371,E2 -28780.371} C_VEL
LIN {X 0,Y 58.553,Z 365.807,A -85,B 0,C 180,E1 -28784.383,E2 -28784.383} C_VEL
LIN {X 0,Y 58.818,Z 365.774,A -85,B 0,C 180,E1 -28793.136,E2 -28793.136} C_VEL
LIN {X 0,Y 59.391,Z 365.707,A -85,B 0,C 180,E1 -28799.998,E2 -28799.998} C_VEL
LIN {X 0,Y 58.817,Z 365.783,A -85,B 0,C 180,E1 -28806.861,E2 -28806.861} C_VEL
LIN {X 0,Y 58.52,Z 365.819,A -85,B 0,C 180,E1 -28816.127,E2 -28816.127} C_VEL
LIN {X 0,Y 58.315,Z 365.838,A -85,B 0,C 180,E1 -28828.819,E2 -28828.819} C_VEL
LIN {X 0,Y 58.844,Z 365.774,A -85,B 0,C 180,E1 -28836.666,E2 -28836.666} C_VEL
LIN {X 0,Y 60.802,Z 365.752,A -85,B 0,C 180,E1 -28848.105,E2 -28848.105} C_VEL
LIN {X 0,Y 60.897,Z 366.569,A -85,B 0,C 180,E1 -28848.984,E2 -28848.984} C_VEL
LIN {X 0,Y 59.626,Z 384.281,A -85,B 0,C 180,E1 -28855.594,E2 -28855.594} C_VEL
LIN {X 0,Y 59.925,Z 399.531,A -85,B 0,C 180,E1 -28862.758,E2 -28862.758} C_VEL
LIN {X 0,Y 61.693,Z 414.23,A -85,B 0,C 180,E1 -28870.888,E2 -28870.888} C_VEL
LIN {X 0,Y 64.473,Z 426.92,A -85,B 0,C 180,E1 -28878.825,E2 -28878.825} C_VEL
LIN {X 0,Y 66.136,Z 432.329,A -85,B 0,C 180,E1 -28882.447,E2 -28882.447} C_VEL
LIN {X 0,Y 66.847,Z 436.017,A -85,B 0,C 180,E1 -28885.483,E2 -28885.483} C_VEL
LIN {X 0,Y 68.432,Z 443.756,A -85,B 0,C 180,E1 -28892.949,E2 -28892.949} C_VEL
LIN {X 0,Y 70.297,Z 449.108,A -85,B 0,C 180,E1 -28898.63,E2 -28898.63} C_VEL
LIN {X 0,Y 69.425,Z 451.478,A -85,B 0,C 180,E1 -28904.665,E2 -28904.665} C_VEL
LIN {X 0,Y 70.568,Z 456.141,A -85,B 0,C 180,E1 -28919.871,E2 -28919.871} C_VEL
LIN {X 0,Y 78.616,Z 460.296,A -85,B 0,C 180,E1 -28935.663,E2 -28935.663} C_VEL
LIN {X 0,Y 79.512,Z 460.548,A -85,B 0,C 180,E1 -28936.752,E2 -28936.752} C_VEL
LIN {X 0,Y 79.881,Z 460.315,A -85,B 0,C 180,E1 -28938.274,E2 -28938.274} C_VEL
LIN {X 0,Y 70.32,Z 450.127,A -85,B 0,C 180,E1 -28948.354,E2 -28948.354} C_VEL
LIN {X 0,Y 63.961,Z 438.609,A -85,B 0,C 180,E1 -28960.755,E2 -28960.755} C_VEL
LIN {X 0,Y 61.549,Z 429.71,A -85,B 0,C 180,E1 -28970.14,E2 -28970.14} C_VEL
LIN {X 0,Y 60.432,Z 417.62,A -85,B 0,C 180,E1 -28981.668,E2 -28981.668} C_VEL
LIN {X 0,Y 61.057,Z 406.538,A -85,B 0,C 180,E1 -28990.782,E2 -28990.782} C_VEL
LIN {X 0,Y 62.837,Z 393.468,A -85,B 0,C 180,E1 -28999.607,E2 -28999.607} C_VEL
LIN {X 0,Y 63.867,Z 386.638,A -85,B 0,C 180,E1 -29003.47,E2 -29003.47} C_VEL
LIN {X 0,Y 60.201,Z 372.918,A -85,B 0,C 180,E1 -29009.811,E2 -29009.811} C_VEL
LIN {X 0,Y 58.689,Z 366.406,A -85,B 0,C 180,E1 -29012.863,E2 -29012.863} C_VEL
LIN {X 0,Y 58.531,Z 365.882,A -85,B 0,C 180,E1 -29013.816,E2 -29013.816} C_VEL
LIN {X 0,Y 58.035,Z 365.874,A -85,B 0,C 180,E1 -29026.605,E2 -29026.605} C_VEL
LIN {X 0,Y 58.043,Z 365.871,A -85,B 0,C 180,E1 -29032.734,E2 -29032.734} C_VEL
LIN {X 0,Y 58.164,Z 365.865,A -85,B 0,C 180,E1 -29037.762,E2 -29037.762} C_VEL
LIN {X 0,Y 58.155,Z 365.858,A -85,B 0,C 180,E1 -29041.086,E2 -29041.086} C_VEL
LIN {X 0,Y 58.53,Z 365.818,A -85,B 0,C 180,E1 -29053.87,E2 -29053.87} C_VEL
LIN {X 0,Y 58.828,Z 365.782,A -85,B 0,C 180,E1 -29063.132,E2 -29063.132} C_VEL
LIN {X 0,Y 59.401,Z 365.707,A -85,B 0,C 180,E1 -29069.994,E2 -29069.994} C_VEL
LIN {X 0,Y 58.827,Z 365.773,A -85,B 0,C 180,E1 -29076.855,E2 -29076.855} C_VEL
LIN {X 0,Y 58.539,Z 365.81,A -85,B 0,C 180,E1 -29086.159,E2 -29086.159} C_VEL
LIN {X 0,Y 58.151,Z 365.865,A -85,B 0,C 180,E1 -29098.902,E2 -29098.902} C_VEL
LIN {X 0,Y 58.157,Z 365.856,A -85,B 0,C 180,E1 -29102.225,E2 -29102.225} C_VEL
LIN {X 0,Y 58.03,Z 365.881,A -85,B 0,C 180,E1 -29107.26,E2 -29107.26} C_VEL
LIN {X 0,Y 58.008,Z 365.881,A -85,B 0,C 180,E1 -29116.62,E2 -29116.62} C_VEL
LIN {X 0,Y 58.028,Z 365.881,A -85,B 0,C 180,E1 -29122.728,E2 -29122.728} C_VEL
LIN {X 0,Y 58.154,Z 365.857,A -85,B 0,C 180,E1 -29127.763,E2 -29127.763} C_VEL
LIN {X 0,Y 58.148,Z 365.866,A -85,B 0,C 180,E1 -29131.086,E2 -29131.086} C_VEL
LIN {X 0,Y 58.553,Z 365.807,A -85,B 0,C 180,E1 -29144.383,E2 -29144.383} C_VEL
LIN {X 0,Y 58.036,Z 365.88,A -85,B 0,C 180,E1 -29148.166,E2 -29148.166} C_VEL
LIN {X 0,Y 56.625,Z 366.054,A -85,B 0,C 180,E1 -29151.862,E2 -29151.862} C_VEL
LIN {X 0,Y 51.911,Z 366.638,A -85,B 0,C 180,E1 -29163.973,E2 -29163.973} C_VEL
LIN {X 0,Y 51.762,Z 366.646,A -85,B 0,C 180,E1 -29165.493,E2 -29165.493} C_VEL
LIN {X 0,Y 51.391,Z 366.703,A -85,B 0,C 180,E1 -29176.831,E2 -29176.831} C_VEL
LIN {X 0,Y 51.5,Z 366.694,A -85,B 0,C 180,E1 -29193.081,E2 -29193.081} C_VEL
LIN {X 0,Y 53.642,Z 366.668,A -85,B 0,C 180,E1 -29208.335,E2 -29208.335} C_VEL
LIN {X 0,Y 53.6,Z 367.946,A -85,B 0,C 180,E1 -29209.562,E2 -29209.562} C_VEL
LIN {X 0,Y 52.589,Z 383.218,A -85,B 0,C 180,E1 -29216.078,E2 -29216.078} C_VEL
LIN {X 0,Y 52.915,Z 397.037,A -85,B 0,C 180,E1 -29223.376,E2 -29223.376} C_VEL
LIN {X 0,Y 54.787,Z 411.514,A -85,B 0,C 180,E1 -29232.269,E2 -29232.269} C_VEL
LIN {X 0,Y 58.032,Z 424.789,A -85,B 0,C 180,E1 -29241.285,E2 -29241.285} C_VEL
LIN {X 0,Y 60.553,Z 432.143,A -85,B 0,C 180,E1 -29246.679,E2 -29246.679} C_VEL
LIN {X 0,Y 62.449,Z 440.252,A -85,B 0,C 180,E1 -29254.848,E2 -29254.848} C_VEL
LIN {X 0,Y 64.424,Z 445.584,A -85,B 0,C 180,E1 -29260.953,E2 -29260.953} C_VEL
LIN {X 0,Y 64.093,Z 450.422,A -85,B 0,C 180,E1 -29276.022,E2 -29276.022} C_VEL
LIN {X 0,Y 70.731,Z 455.272,A -85,B 0,C 180,E1 -29294.076,E2 -29294.076} C_VEL
LIN {X 0,Y 72.198,Z 455.625,A -85,B 0,C 180,E1 -29297.049,E2 -29297.049} C_VEL
LIN {X 0,Y 62.87,Z 444.936,A -85,B 0,C 180,E1 -29307.93,E2 -29307.93} C_VEL
LIN {X 0,Y 57.239,Z 434.008,A -85,B 0,C 180,E1 -29320.268,E2 -29320.268} C_VEL
LIN {X 0,Y 54.677,Z 424.435,A -85,B 0,C 180,E1 -29330.756,E2 -29330.756} C_VEL
LIN {X 0,Y 53.98,Z 410.502,A -85,B 0,C 180,E1 -29344.669,E2 -29344.669} C_VEL
LIN {X 0,Y 55.173,Z 396.903,A -85,B 0,C 180,E1 -29355.707,E2 -29355.707} C_VEL
LIN {X 0,Y 56.763,Z 386.767,A -85,B 0,C 180,E1 -29362.448,E2 -29362.448} C_VEL
LIN {X 0,Y 52.911,Z 372.661,A -85,B 0,C 180,E1 -29369.6,E2 -29369.6} C_VEL
LIN {X 0,Y 51.667,Z 367.306,A -85,B 0,C 180,E1 -29372.427,E2 -29372.427} C_VEL
LIN {X 0,Y 51.441,Z 366.722,A -85,B 0,C 180,E1 -29374.177,E2 -29374.177} C_VEL
LIN {X 0,Y 51.003,Z 366.749,A -85,B 0,C 180,E1 -29386.442,E2 -29386.442} C_VEL
LIN {X 0,Y 51.058,Z 366.748,A -85,B 0,C 180,E1 -29396.584,E2 -29396.584} C_VEL
LIN {X 0,Y 51.029,Z 366.753,A -85,B 0,C 180,E1 -29405.588,E2 -29405.588} C_VEL
LIN {X 0,Y 51.471,Z 366.698,A -85,B 0,C 180,E1 -29414.145,E2 -29414.145} C_VEL
LIN {X 0,Y 51.701,Z 366.668,A -85,B 0,C 180,E1 -29422.18,E2 -29422.18} C_VEL
LIN {X 0,Y 52.285,Z 366.592,A -85,B 0,C 180,E1 -29429.993,E2 -29429.993} C_VEL
LIN {X 0,Y 51.702,Z 366.662,A -85,B 0,C 180,E1 -29437.805,E2 -29437.805} C_VEL
LIN {X 0,Y 51.404,Z 366.701,A -85,B 0,C 180,E1 -29446.848,E2 -29446.848} C_VEL
LIN {X 0,Y 51.026,Z 366.745,A -85,B 0,C 180,E1 -29454.398,E2 -29454.398} C_VEL
LIN {X 0,Y 51.028,Z 366.749,A -85,B 0,C 180,E1 -29464.268,E2 -29464.268} C_VEL
LIN {X 0,Y 50.975,Z 366.758,A -85,B 0,C 180,E1 -29476.418,E2 -29476.418} C_VEL
LIN {X 0,Y 51.046,Z 366.743,A -85,B 0,C 180,E1 -29486.581,E2 -29486.581} C_VEL
LIN {X 0,Y 51.022,Z 366.745,A -85,B 0,C 180,E1 -29495.589,E2 -29495.589} C_VEL
LIN {X 0,Y 51.477,Z 366.689,A -85,B 0,C 180,E1 -29504.152,E2 -29504.152} C_VEL
LIN {X 0,Y 51.694,Z 366.662,A -85,B 0,C 180,E1 -29512.184,E2 -29512.184} C_VEL
LIN {X 0,Y 52.275,Z 366.592,A -85,B 0,C 180,E1 -29519.998,E2 -29519.998} C_VEL
LIN {X 0,Y 51.762,Z 366.646,A -85,B 0,C 180,E1 -29525.493,E2 -29525.493} C_VEL
LIN {X 0,Y 51.227,Z 366.725,A -85,B 0,C 180,E1 -29529.802,E2 -29529.802} C_VEL
LIN {X 0,Y 49.61,Z 366.935,A -85,B 0,C 180,E1 -29536.259,E2 -29536.259} C_VEL
LIN {X 0,Y 46.366,Z 367.333,A -85,B 0,C 180,E1 -29547.676,E2 -29547.676} C_VEL
LIN {X 0,Y 45.111,Z 367.49,A -85,B 0,C 180,E1 -29560.461,E2 -29560.461} C_VEL
LIN {X 0,Y 45.387,Z 367.446,A -85,B 0,C 180,E1 -29563.032,E2 -29563.032} C_VEL
LIN {X 0,Y 46.387,Z 367.451,A -85,B 0,C 180,E1 -29568.42,E2 -29568.42} C_VEL
LIN {X 0,Y 46.426,Z 368.408,A -85,B 0,C 180,E1 -29569.833,E2 -29569.833} C_VEL
LIN {X 0,Y 45.609,Z 385.336,A -85,B 0,C 180,E1 -29578.673,E2 -29578.673} C_VEL
LIN {X 0,Y 46.531,Z 400.311,A -85,B 0,C 180,E1 -29588.226,E2 -29588.226} C_VEL
LIN {X 0,Y 49.241,Z 414.211,A -85,B 0,C 180,E1 -29598.099,E2 -29598.099} C_VEL
LIN {X 0,Y 53.588,Z 427.398,A -85,B 0,C 180,E1 -29608.128,E2 -29608.128} C_VEL
LIN {X 0,Y 54.626,Z 429.864,A -85,B 0,C 180,E1 -29610.007,E2 -29610.007} C_VEL
LIN {X 0,Y 57.073,Z 437.877,A -85,B 0,C 180,E1 -29618.681,E2 -29618.681} C_VEL
LIN {X 0,Y 58.299,Z 440.776,A -85,B 0,C 180,E1 -29622.12,E2 -29622.12} C_VEL
LIN {X 0,Y 58.7,Z 441.948,A -85,B 0,C 180,E1 -29623.861,E2 -29623.861} C_VEL
LIN {X 0,Y 58.925,Z 446.281,A -85,B 0,C 180,E1 -29638.501,E2 -29638.501} C_VEL
LIN {X 0,Y 63.207,Z 449.811,A -85,B 0,C 180,E1 -29651.854,E2 -29651.854} C_VEL
LIN {X 0,Y 64.729,Z 450.38,A -85,B 0,C 180,E1 -29655.576,E2 -29655.576} C_VEL
LIN {X 0,Y 55.59,Z 439.155,A -85,B 0,C 180,E1 -29667.501,E2 -29667.501} C_VEL
LIN {X 0,Y 50.088,Z 427.318,A -85,B 0,C 180,E1 -29681.599,E2 -29681.599} C_VEL
LIN {X 0,Y 47.482,Z 413.001,A -85,B 0,C 180,E1 -29697.882,E2 -29697.882} C_VEL
LIN {X 0,Y 47.738,Z 401.195,A -85,B 0,C 180,E1 -29709.536,E2 -29709.536} C_VEL
LIN {X 0,Y 49.308,Z 388.519,A -85,B 0,C 180,E1 -29719.789,E2 -29719.789} C_VEL
LIN {X 0,Y 49.498,Z 386.235,A -85,B 0,C 180,E1 -29721.338,E2 -29721.338} C_VEL
LIN {X 0,Y 45.095,Z 370.053,A -85,B 0,C 180,E1 -29730.475,E2 -29730.475} C_VEL
LIN {X 0,Y 44.568,Z 368.002,A -85,B 0,C 180,E1 -29732.033,E2 -29732.033} C_VEL
LIN {X 0,Y 44.428,Z 367.601,A -85,B 0,C 180,E1 -29733.65,E2 -29733.65} C_VEL
LIN {X 0,Y 43.983,Z 367.629,A -85,B 0,C 180,E1 -29739.732,E2 -29739.732} C_VEL
LIN {X 0,Y 43.852,Z 367.638,A -85,B 0,C 180,E1 -29753.261,E2 -29753.261} C_VEL
LIN {X 0,Y 43.849,Z 367.639,A -85,B 0,C 180,E1 -29761.251,E2 -29761.251} C_VEL
LIN {X 0,Y 44.236,Z 367.592,A -85,B 0,C 180,E1 -29772.42,E2 -29772.42} C_VEL
LIN {X 0,Y 44.551,Z 367.553,A -85,B 0,C 180,E1 -29780.915,E2 -29780.915} C_VEL
LIN {X 0,Y 45.16,Z 367.479,A -85,B 0,C 180,E1 -29789.992,E2 -29789.992} C_VEL
LIN {X 0,Y 44.554,Z 367.556,A -85,B 0,C 180,E1 -29799.067,E2 -29799.067} C_VEL
LIN {X 0,Y 44.195,Z 367.604,A -85,B 0,C 180,E1 -29808.536,E2 -29808.536} C_VEL
LIN {X 0,Y 43.843,Z 367.647,A -85,B 0,C 180,E1 -29818.734,E2 -29818.734} C_VEL
LIN {X 0,Y 43.798,Z 367.645,A -85,B 0,C 180,E1 -29829.919,E2 -29829.919} C_VEL
LIN {X 0,Y 43.837,Z 367.65,A -85,B 0,C 180,E1 -29843.269,E2 -29843.269} C_VEL
LIN {X 0,Y 43.839,Z 367.649,A -85,B 0,C 180,E1 -29851.25,E2 -29851.25} C_VEL
LIN {X 0,Y 44.252,Z 367.593,A -85,B 0,C 180,E1 -29862.315,E2 -29862.315} C_VEL
LIN {X 0,Y 44.546,Z 367.556,A -85,B 0,C 180,E1 -29870.92,E2 -29870.92} C_VEL
LIN {X 0,Y 45.15,Z 367.479,A -85,B 0,C 180,E1 -29879.998,E2 -29879.998} C_VEL
LIN {X 0,Y 44.541,Z 367.553,A -85,B 0,C 180,E1 -29889.076,E2 -29889.076} C_VEL
LIN {X 0,Y 44.198,Z 367.595,A -85,B 0,C 180,E1 -29898.541,E2 -29898.541} C_VEL
LIN {X 0,Y 44.094,Z 367.608,A -85,B 0,C 180,E1 -29908.563,E2 -29908.563} C_VEL
LIN {X 0,Y 45.387,Z 367.446,A -85,B 0,C 180,E1 -29923.032,E2 -29923.032} C_VEL
LIN {X 0,Y 45.231,Z 368.036,A -85,B 0,C 180,E1 -29926.009,E2 -29926.009} C_VEL
LIN {X 0,Y 43.92,Z 369.954,A -85,B 0,C 180,E1 -29929.302,E2 -29929.302} C_VEL
LIN {X 0,Y 41.46,Z 373.434,A -85,B 0,C 180,E1 -29932.607,E2 -29932.607} C_VEL
LIN {X 0,Y 39.754,Z 376.682,A -85,B 0,C 180,E1 -29934.987,E2 -29934.987} C_VEL
LIN {X 0,Y 38.732,Z 380.711,A -85,B 0,C 180,E1 -29937.794,E2 -29937.794} C_VEL
LIN {X 0,Y 38.723,Z 389.054,A -85,B 0,C 180,E1 -29943.69,E2 -29943.69} C_VEL
LIN {X 0,Y 39.161,Z 393.103,A -85,B 0,C 180,E1 -29946.668,E2 -29946.668} C_VEL
LIN {X 0,Y 41.613,Z 407.319,A -85,B 0,C 180,E1 -29957.822,E2 -29957.822} C_VEL
LIN {X 0,Y 45.945,Z 420.848,A -85,B 0,C 180,E1 -29968.912,E2 -29968.912} C_VEL
LIN {X 0,Y 49.4,Z 428.567,A -85,B 0,C 180,E1 -29975.23,E2 -29975.23} C_VEL
LIN {X 0,Y 52.885,Z 437.156,A -85,B 0,C 180,E1 -29985.421,E2 -29985.421} C_VEL
LIN {X 0,Y 53.131,Z 438.193,A -85,B 0,C 180,E1 -29987.568,E2 -29987.568} C_VEL
LIN {X 0,Y 56.023,Z 443.896,A -85,B 0,C 180,E1 -30008.855,E2 -30008.855} C_VEL
LIN {X 0,Y 57.752,Z 444.981,A -85,B 0,C 180,E1 -30013.103,E2 -30013.103} C_VEL
LIN {X 0,Y 55.578,Z 442.57,A -85,B 0,C 180,E1 -30015.937,E2 -30015.937} C_VEL
LIN {X 0,Y 47.57,Z 431.336,A -85,B 0,C 180,E1 -30028.865,E2 -30028.865} C_VEL
LIN {X 0,Y 43.378,Z 421.545,A -85,B 0,C 180,E1 -30041.095,E2 -30041.095} C_VEL
LIN {X 0,Y 41.115,Z 408.254,A -85,B 0,C 180,E1 -30057.553,E2 -30057.553} C_VEL
LIN {X 0,Y 41.369,Z 395.667,A -85,B 0,C 180,E1 -30071.021,E2 -30071.021} C_VEL
LIN {X 0,Y 42.469,Z 386.239,A -85,B 0,C 180,E1 -30079.331,E2 -30079.331} C_VEL
LIN {X 0,Y 38.133,Z 371.058,A -85,B 0,C 180,E1 -30089.079,E2 -30089.079} C_VEL
LIN {X 0,Y 37.572,Z 368.846,A -85,B 0,C 180,E1 -30091.037,E2 -30091.037} C_VEL
LIN {X 0,Y 37.237,Z 368.465,A -85,B 0,C 180,E1 -30094.49,E2 -30094.49} C_VEL
LIN {X 0,Y 36.749,Z 368.532,A -85,B 0,C 180,E1 -30109.91,E2 -30109.91} C_VEL
LIN {X 0,Y 36.731,Z 368.526,A -85,B 0,C 180,E1 -30114.958,E2 -30114.958} C_VEL
LIN {X 0,Y 37.062,Z 368.484,A -85,B 0,C 180,E1 -30131.479,E2 -30131.479} C_VEL
LIN {X 0,Y 37.343,Z 368.448,A -85,B 0,C 180,E1 -30139.142,E2 -30139.142} C_VEL
LIN {X 0,Y 38.018,Z 368.367,A -85,B 0,C 180,E1 -30149.99,E2 -30149.99} C_VEL
LIN {X 0,Y 37.351,Z 368.458,A -85,B 0,C 180,E1 -30160.835,E2 -30160.835} C_VEL
LIN {X 0,Y 37.081,Z 368.49,A -85,B 0,C 180,E1 -30168.608,E2 -30168.608} C_VEL
LIN {X 0,Y 36.719,Z 368.532,A -85,B 0,C 180,E1 -30185.031,E2 -30185.031} C_VEL
LIN {X 0,Y 36.719,Z 368.526,A -85,B 0,C 180,E1 -30190.036,E2 -30190.036} C_VEL
LIN {X 0,Y 36.718,Z 368.526,A -85,B 0,C 180,E1 -30199.945,E2 -30199.945} C_VEL
LIN {X 0,Y 36.717,Z 368.531,A -85,B 0,C 180,E1 -30204.951,E2 -30204.951} C_VEL
LIN {X 0,Y 37.075,Z 368.49,A -85,B 0,C 180,E1 -30221.376,E2 -30221.376} C_VEL
LIN {X 0,Y 37.344,Z 368.459,A -85,B 0,C 180,E1 -30229.149,E2 -30229.149} C_VEL
LIN {X 0,Y 38.009,Z 368.368,A -85,B 0,C 180,E1 -30239.997,E2 -30239.997} C_VEL
LIN {X 0,Y 37.34,Z 368.449,A -85,B 0,C 180,E1 -30250.846,E2 -30250.846} C_VEL
LIN {X 0,Y 36.958,Z 368.504,A -85,B 0,C 180,E1 -30262.35,E2 -30262.35} C_VEL
LIN {X 0,Y 38.168,Z 368.349,A -85,B 0,C 180,E1 -30282.578,E2 -30282.578} C_VEL
LIN {X 0,Y 39.306,Z 368.421,A -85,B 0,C 180,E1 -30289.432,E2 -30289.432} C_VEL
LIN {X 0,Y 39.18,Z 369.694,A -85,B 0,C 180,E1 -30291.122,E2 -30291.122} C_VEL
LIN {X 0,Y 38.649,Z 384.185,A -85,B 0,C 180,E1 -30300.184,E2 -30300.184} C_VEL
LIN {X 0,Y 39.161,Z 393.103,A -85,B 0,C 180,E1 -30306.668,E2 -30306.668} C_VEL
LIN {X 0,Y 39.228,Z 398.227,A -85,B 0,C 180,E1 -30310.966,E2 -30310.966} C_VEL
LIN {X 0,Y 38.393,Z 406.135,A -85,B 0,C 180,E1 -30319.734,E2 -30319.734} C_VEL
LIN {X 0,Y 38.678,Z 413.741,A -85,B 0,C 180,E1 -30329.314,E2 -30329.314} C_VEL
LIN {X 0,Y 40.231,Z 418.403,A -85,B 0,C 180,E1 -30334.167,E2 -30334.167} C_VEL
LIN {X 0,Y 44.415,Z 426.507,A -85,B 0,C 180,E1 -30340.942,E2 -30340.942} C_VEL
LIN {X 0,Y 47.759,Z 433.345,A -85,B 0,C 180,E1 -30349.449,E2 -30349.449} C_VEL
LIN {X 0,Y 47.961,Z 434.202,A -85,B 0,C 180,E1 -30351.711,E2 -30351.711} C_VEL
LIN {X 0,Y 50.189,Z 438.307,A -85,B 0,C 180,E1 -30368.012,E2 -30368.012} C_VEL
LIN {X 0,Y 50.217,Z 438.066,A -85,B 0,C 180,E1 -30371.932,E2 -30371.932} C_VEL
LIN {X 0,Y 41.344,Z 425.783,A -85,B 0,C 180,E1 -30386.467,E2 -30386.467} C_VEL
LIN {X 0,Y 36.792,Z 415.268,A -85,B 0,C 180,E1 -30400.474,E2 -30400.474} C_VEL
LIN {X 0,Y 34.707,Z 403.018,A -85,B 0,C 180,E1 -30417.101,E2 -30417.101} C_VEL
LIN {X 0,Y 35.135,Z 389.529,A -85,B 0,C 180,E1 -30433.008,E2 -30433.008} C_VEL
LIN {X 0,Y 35.458,Z 385.966,A -85,B 0,C 180,E1 -30436.557,E2 -30436.557} C_VEL
LIN {X 0,Y 30.657,Z 369.837,A -85,B 0,C 180,E1 -30448.995,E2 -30448.995} C_VEL
LIN {X 0,Y 30.391,Z 369.278,A -85,B 0,C 180,E1 -30451.269,E2 -30451.269} C_VEL
LIN {X 0,Y 29.636,Z 369.283,A -85,B 0,C 180,E1 -30465.357,E2 -30465.357} C_VEL
LIN {X 0,Y 29.502,Z 369.296,A -85,B 0,C 180,E1 -30481.533,E2 -30481.533} C_VEL
LIN {X 0,Y 29.869,Z 369.261,A -85,B 0,C 180,E1 -30490.26,E2 -30490.26} C_VEL
LIN {X 0,Y 30.116,Z 369.24,A -85,B 0,C 180,E1 -30496.492,E2 -30496.492} C_VEL
LIN {X 0,Y 30.835,Z 369.171,A -85,B 0,C 180,E1 -30509.988,E2 -30509.988} C_VEL
LIN {X 0,Y 30.128,Z 369.237,A -85,B 0,C 180,E1 -30523.477,E2 -30523.477} C_VEL
LIN {X 0,Y 29.89,Z 369.262,A -85,B 0,C 180,E1 -30529.848,E2 -30529.848} C_VEL
LIN {X 0,Y 29.507,Z 369.297,A -85,B 0,C 180,E1 -30538.434,E2 -30538.434} C_VEL
LIN {X 0,Y 29.536,Z 369.295,A -85,B 0,C 180,E1 -30555.53,E2 -30555.53} C_VEL
LIN {X 0,Y 29.504,Z 369.298,A -85,B 0,C 180,E1 -30571.544,E2 -30571.544} C_VEL
LIN {X 0,Y 29.884,Z 369.262,A -85,B 0,C 180,E1 -30580.132,E2 -30580.132} C_VEL
LIN {X 0,Y 30.121,Z 369.238,A -85,B 0,C 180,E1 -30586.504,E2 -30586.504} C_VEL
LIN {X 0,Y 30.827,Z 369.172,A -85,B 0,C 180,E1 -30599.997,E2 -30599.997} C_VEL
LIN {X 0,Y 30.134,Z 369.239,A -85,B 0,C 180,E1 -30613.483,E2 -30613.483} C_VEL
LIN {X 0,Y 29.974,Z 369.252,A -85,B 0,C 180,E1 -30620.339,E2 -30620.339} C_VEL
LIN {X 0,Y 31.76,Z 369.12,A -85,B 0,C 180,E1 -30648.421,E2 -30648.421} C_VEL
LIN {X 0,Y 32.09,Z 369.41,A -85,B 0,C 180,E1 -30651.19,E2 -30651.19} C_VEL
LIN {X 0,Y 31.994,Z 371.067,A -85,B 0,C 180,E1 -30653.242,E2 -30653.242} C_VEL
LIN {X 0,Y 31.965,Z 386.621,A -85,B 0,C 180,E1 -30665.667,E2 -30665.667} C_VEL
LIN {X 0,Y 34.485,Z 402.158,A -85,B 0,C 180,E1 -30679.698,E2 -30679.698} C_VEL
LIN {X 0,Y 38.81,Z 415.116,A -85,B 0,C 180,E1 -30691.284,E2 -30691.284} C_VEL
LIN {X 0,Y 40.231,Z 418.403,A -85,B 0,C 180,E1 -30694.167,E2 -30694.167} C_VEL
LIN {X 0,Y 41.337,Z 421.466,A -85,B 0,C 180,E1 -30697.494,E2 -30697.494} C_VEL
LIN {X 0,Y 42.082,Z 424.904,A -85,B 0,C 180,E1 -30703.11,E2 -30703.11} C_VEL
LIN {X 0,Y 42.661,Z 428.314,A -85,B 0,C 180,E1 -30711.256,E2 -30711.256} C_VEL
LIN {X 0,Y 43.241,Z 430.391,A -85,B 0,C 180,E1 -30718.16,E2 -30718.16} C_VEL
LIN {X 0,Y 44.56,Z 432.405,A -85,B 0,C 180,E1 -30727.949,E2 -30727.949} C_VEL
LIN {X 0,Y 36.32,Z 421.434,A -85,B 0,C 180,E1 -30741.032,E2 -30741.032} C_VEL
LIN {X 0,Y 30.367,Z 408.28,A -85,B 0,C 180,E1 -30759.691,E2 -30759.691} C_VEL
LIN {X 0,Y 28.579,Z 398.481,A -85,B 0,C 180,E1 -30774.712,E2 -30774.712} C_VEL
LIN {X 0,Y 28.62,Z 385.67,A -85,B 0,C 180,E1 -30792.234,E2 -30792.234} C_VEL
LIN {X 0,Y 23.69,Z 370.295,A -85,B 0,C 180,E1 -30806.332,E2 -30806.332} C_VEL
LIN {X 0,Y 23.35,Z 369.732,A -85,B 0,C 180,E1 -30809.326,E2 -30809.326} C_VEL
LIN {X 0,Y 22.704,Z 369.694,A -85,B 0,C 180,E1 -30818.257,E2 -30818.257} C_VEL
LIN {X 0,Y 22.242,Z 369.707,A -85,B 0,C 180,E1 -30830.785,E2 -30830.785} C_VEL
LIN {X 0,Y 22.818,Z 369.689,A -85,B 0,C 180,E1 -30852.044,E2 -30852.044} C_VEL
LIN {X 0,Y 23.602,Z 369.666,A -85,B 0,C 180,E1 -30869.985,E2 -30869.985} C_VEL
LIN {X 0,Y 22.842,Z 369.689,A -85,B 0,C 180,E1 -30887.903,E2 -30887.903} C_VEL
LIN {X 0,Y 22.195,Z 369.709,A -85,B 0,C 180,E1 -30909.273,E2 -30909.273} C_VEL
LIN {X 0,Y 22.193,Z 369.709,A -85,B 0,C 180,E1 -30920.696,E2 -30920.696} C_VEL
LIN {X 0,Y 22.836,Z 369.689,A -85,B 0,C 180,E1 -30942.071,E2 -30942.071} C_VEL
LIN {X 0,Y 23.597,Z 369.666,A -85,B 0,C 180,E1 -30959.995,E2 -30959.995} C_VEL
LIN {X 0,Y 22.906,Z 369.687,A -85,B 0,C 180,E1 -30977.863,E2 -30977.863} C_VEL
LIN {X 0,Y 24.956,Z 369.774,A -85,B 0,C 180,E1 -31012.406,E2 -31012.406} C_VEL
LIN {X 0,Y 24.974,Z 370.763,A -85,B 0,C 180,E1 -31015.156,E2 -31015.156} C_VEL
LIN {X 0,Y 25.544,Z 386.889,A -85,B 0,C 180,E1 -31031.985,E2 -31031.985} C_VEL
LIN {X 0,Y 29.179,Z 402.241,A -85,B 0,C 180,E1 -31048.327,E2 -31048.327} C_VEL
LIN {X 0,Y 34.555,Z 414.934,A -85,B 0,C 180,E1 -31060.262,E2 -31060.262} C_VEL
LIN {X 0,Y 39.879,Z 424.172,A -85,B 0,C 180,E1 -31067.973,E2 -31067.973} C_VEL
LIN {X 0,Y 42.986,Z 429.415,A -85,B 0,C 180,E1 -31074.377,E2 -31074.377} C_VEL
LIN {X 0,Y 43.241,Z 430.391,A -85,B 0,C 180,E1 -31078.16,E2 -31078.16} C_VEL
LIN {X 0,Y 42.978,Z 430.415,A -85,B 0,C 180,E1 -31080.575,E2 -31080.575} C_VEL
LIN {X 0,Y 41.91,Z 429.408,A -85,B 0,C 180,E1 -31083.346,E2 -31083.346} C_VEL
LIN {X 0,Y 39.806,Z 427.04,A -85,B 0,C 180,E1 -31086.368,E2 -31086.368} C_VEL
LIN {X 0,Y 31.413,Z 416.176,A -85,B 0,C 180,E1 -31094.649,E2 -31094.649} C_VEL
LIN {X 0,Y 24.758,Z 402.848,A -85,B 0,C 180,E1 -31114.803,E2 -31114.803} C_VEL
LIN {X 0,Y 22.239,Z 390.321,A -85,B 0,C 180,E1 -31136.526,E2 -31136.526} C_VEL
LIN {X 0,Y 22.157,Z 385.608,A -85,B 0,C 180,E1 -31144.507,E2 -31144.507} C_VEL
LIN {X 0,Y 16.78,Z 370.352,A -85,B 0,C 180,E1 -31161.492,E2 -31161.492} C_VEL
LIN {X 0,Y 16.376,Z 369.803,A -85,B 0,C 180,E1 -31165.422,E2 -31165.422} C_VEL
LIN {X 0,Y 15.286,Z 369.803,A -85,B 0,C 180,E1 -31206.877,E2 -31206.877} C_VEL
LIN {X 0,Y 16.267,Z 369.803,A -85,B 0,C 180,E1 -31229.978,E2 -31229.978} C_VEL
LIN {X 0,Y 15.287,Z 369.803,A -85,B 0,C 180,E1 -31253.133,E2 -31253.133} C_VEL
LIN {X 0,Y 15.107,Z 369.803,A -85,B 0,C 180,E1 -31257.696,E2 -31257.696} C_VEL
LIN {X 0,Y 15.104,Z 369.803,A -85,B 0,C 180,E1 -31292.261,E2 -31292.261} C_VEL
LIN {X 0,Y 15.282,Z 369.803,A -85,B 0,C 180,E1 -31296.827,E2 -31296.827} C_VEL
LIN {X 0,Y 16.269,Z 369.803,A -85,B 0,C 180,E1 -31319.993,E2 -31319.993} C_VEL
LIN {X 0,Y 15.668,Z 369.803,A -85,B 0,C 180,E1 -31346.643,E2 -31346.643} C_VEL
LIN {X 0,Y 17.892,Z 369.927,A -85,B 0,C 180,E1 -31376.545,E2 -31376.545} C_VEL
LIN {X 0,Y 18.007,Z 371.226,A -85,B 0,C 180,E1 -31380.458,E2 -31380.458} C_VEL
LIN {X 0,Y 19.614,Z 386.676,A -85,B 0,C 180,E1 -31402.025,E2 -31402.025} C_VEL
LIN {X 0,Y 24.783,Z 402.026,A -85,B 0,C 180,E1 -31420.224,E2 -31420.224} C_VEL
LIN {X 0,Y 31.974,Z 415.491,A -85,B 0,C 180,E1 -31432.133,E2 -31432.133} C_VEL
LIN {X 0,Y 36.641,Z 422.426,A -85,B 0,C 180,E1 -31437.111,E2 -31437.111} C_VEL
LIN {X 0,Y 38.449,Z 425.102,A -85,B 0,C 180,E1 -31440.187,E2 -31440.187} C_VEL
LIN {X 0,Y 38.858,Z 425.789,A -85,B 0,C 180,E1 -31442.872,E2 -31442.872} C_VEL
LIN {X 0,Y 36.416,Z 422.947,A -85,B 0,C 180,E1 -31446.583,E2 -31446.583} C_VEL
LIN {X 0,Y 31.413,Z 416.176,A -85,B 0,C 180,E1 -31454.649,E2 -31454.649} C_VEL
LIN {X 0,Y 28.501,Z 411.692,A -85,B 0,C 180,E1 -31459.232,E2 -31459.232} C_VEL
LIN {X 0,Y 23.548,Z 403.564,A -85,B 0,C 180,E1 -31465.029,E2 -31465.029} C_VEL
LIN {X 0,Y 19.829,Z 396.722,A -85,B 0,C 180,E1 -31470.589,E2 -31470.589} C_VEL
LIN {X 0,Y 17.687,Z 391.606,A -85,B 0,C 180,E1 -31477.638,E2 -31477.638} C_VEL
LIN {X 0,Y 17.206,Z 389.899,A -85,B 0,C 180,E1 -31480.878,E2 -31480.878} C_VEL
LIN {X 0,Y 16.372,Z 385.159,A -85,B 0,C 180,E1 -31491.036,E2 -31491.036} C_VEL
LIN {X 0,Y 11.503,Z 373.782,A -85,B 0,C 180,E1 -31503.049,E2 -31503.049} C_VEL
LIN {X 0,Y 10.154,Z 370.098,A -85,B 0,C 180,E1 -31509.899,E2 -31509.899} C_VEL
LIN {X 0,Y 9.479,Z 369.803,A -85,B 0,C 180,E1 -31516.213,E2 -31516.213} C_VEL
LIN {X 0,Y 7.91,Z 369.803,A -85,B 0,C 180,E1 -31562.714,E2 -31562.714} C_VEL
LIN {X 0,Y 8.702,Z 369.803,A -85,B 0,C 180,E1 -31589.958,E2 -31589.958} C_VEL
LIN {X 0,Y 7.781,Z 369.803,A -85,B 0,C 180,E1 -31615.376,E2 -31615.376} C_VEL
LIN {X 0,Y 7.777,Z 369.803,A -85,B 0,C 180,E1 -31654.543,E2 -31654.543} C_VEL
LIN {X 0,Y 8.701,Z 369.803,A -85,B 0,C 180,E1 -31679.988,E2 -31679.988} C_VEL
LIN {X 0,Y 8.688,Z 369.803,A -85,B 0,C 180,E1 -31716.082,E2 -31716.082} C_VEL
LIN {X 0,Y 11.195,Z 369.995,A -85,B 0,C 180,E1 -31747.245,E2 -31747.245} C_VEL
LIN {X 0,Y 11.445,Z 371.478,A -85,B 0,C 180,E1 -31752.153,E2 -31752.153} C_VEL
LIN {X 0,Y 15.306,Z 387.654,A -85,B 0,C 180,E1 -31781.512,E2 -31781.512} C_VEL
LIN {X 0,Y 22.261,Z 402.323,A -85,B 0,C 180,E1 -31796.729,E2 -31796.729} C_VEL
LIN {X 0,Y 27.506,Z 410.83,A -85,B 0,C 180,E1 -31802.491,E2 -31802.491} C_VEL
LIN {X 0,Y 26.499,Z 409.588,A -85,B 0,C 180,E1 -31807.29,E2 -31807.29} C_VEL
LIN {X 0,Y 19.946,Z 397.983,A -85,B 0,C 180,E1 -31825.077,E2 -31825.077} C_VEL
LIN {X 0,Y 17.206,Z 389.899,A -85,B 0,C 180,E1 -31840.878,E2 -31840.878} C_VEL
LIN {X 0,Y 16.137,Z 387.125,A -85,B 0,C 180,E1 -31844.6,E2 -31844.6} C_VEL
LIN {X 0,Y 13.71,Z 383.187,A -85,B 0,C 180,E1 -31844.868,E2 -31844.868} C_VEL
LIN {X 0,Y 8.167,Z 375.481,A -85,B 0,C 180,E1 -31831.402,E2 -31831.402} C_VEL
LIN {X 0,Y 6.29,Z 371.788,A -85,B 0,C 180,E1 -31826.807,E2 -31826.807} C_VEL
LIN {X 0,Y 5.181,Z 369.803,A -85,B 0,C 180,E1 -31828.827,E2 -31828.827} C_VEL
LIN {X 0,Y 1.044,Z 369.803,A -85,B 0,C 180,E1 -31860.102,E2 -31860.102} C_VEL
LIN {X 0,Y 0.361,Z 369.803,A -85,B 0,C 180,E1 -31948.987,E2 -31948.987} C_VEL
LIN {X 0,Y 0.352,Z 369.803,A -85,B 0,C 180,E1 -32039.697,E2 -32039.697} C_VEL
LIN {X 0,Y 3.295,Z 369.803,A -85,B 0,C 180,E1 -32130.111,E2 -32130.111} C_VEL
LIN {X 0,Y 5.869,Z 369.972,A -85,B 0,C 180,E1 -32142.502,E2 -32142.502} C_VEL
LIN {X 0,Y 13.391,Z 387.624,A -85,B 0,C 180,E1 -32169.285,E2 -32169.285} C_VEL
LIN {X 0,Y 13.931,Z 388.69,A -85,B 0,C 180,E1 -32170.03,E2 -32170.03} C_VEL
LIN {X 0,Y 13.568,Z 387.535,A -85,B 0,C 180,E1 -32179.658,E2 -32179.658} C_VEL
LIN {X 0,Y 12.163,Z 384.027,A -85,B 0,C 180,E1 -32187.203,E2 -32187.203} C_VEL
LIN {X 0,Y 6.29,Z 371.788,A -85,B 0,C 180,E1 -32186.807,E2 -32186.807} C_VEL
LIN {X 0,Y 2.492,Z 372.594,A -85,B 0,C 180,E1 -32194.029,E2 -32194.029} C_VEL
LIN {X 0,Y 2.492,Z 600,A -85,B 0,C 180,E1 -32194.029,E2 -32194.029} C_VEL
LIN {X 0,Y 2.492,Z 600,A -85,B 0,C 180,E1 -32194.029,E2 -32194.029}

QRS_NEXT_CUT()

QRS_NEXT()
QRS_HOME()

END
